   LIN {X -2.321, Y 6.996, Z 4.250} C_DIS
   LIN {X -2.151, Y 7.892, Z 4.250} C_DIS
   LIN {X -2.103, Y 8.164, Z 4.250} C_DIS
   LIN {X -1.982, Y 8.852, Z 4.250} C_DIS
   LIN {X -1.964, Y 8.960, Z 4.250} C_DIS
   LIN {X -1.822, Y 9.845, Z 4.250} C_DIS
   LIN {X -1.804, Y 9.955, Z 4.250} C_DIS
   LIN {X -1.672, Y 10.861, Z 4.250} C_DIS
   LIN {X -1.586, Y 11.505, Z 4.250} C_DIS
   LIN {X -1.538, Y 11.861, Z 4.250} C_DIS
   LIN {X -1.420, Y 12.858, Z 4.250} C_DIS
   LIN {X -1.315, Y 13.857, Z 4.250} C_DIS
   LIN {X -1.225, Y 14.841, Z 4.250} C_DIS
   LIN {X -1.150, Y 15.814, Z 4.250} C_DIS
   LIN {X -1.140, Y 15.955, Z 4.250} C_DIS
   LIN {X -1.088, Y 16.783, Z 4.250} C_DIS
   LIN {X -1.080, Y 16.934, Z 4.250} C_DIS
   LIN {X -1.038, Y 17.778, Z 4.250} C_DIS
   LIN {X -1.032, Y 17.929, Z 4.250} C_DIS
   LIN {X -1.001, Y 18.785, Z 4.250} C_DIS
   LIN {X -0.981, Y 19.646, Z 4.250} C_DIS
   LIN {X -0.976, Y 19.937, Z 4.250} C_DIS
   LIN {X -0.968, Y 20.790, Z 4.250} C_DIS
   LIN {X -0.969, Y 20.932, Z 4.250} C_DIS
   LIN {X -0.973, Y 21.776, Z 4.250} C_DIS
   LIN {X -0.975, Y 21.917, Z 4.250} C_DIS
   LIN {X -0.991, Y 22.780, Z 4.250} C_DIS
   LIN {X -0.995, Y 22.916, Z 4.250} C_DIS
   LIN {X -1.023, Y 23.792, Z 4.250} C_DIS
   LIN {X -1.029, Y 23.927, Z 4.250} C_DIS
   LIN {X -1.069, Y 24.801, Z 4.250} C_DIS
   LIN {X -1.077, Y 24.932, Z 4.250} C_DIS
   LIN {X -1.128, Y 25.791, Z 4.250} C_DIS
   LIN {X -1.137, Y 25.919, Z 4.250} C_DIS
   LIN {X -1.201, Y 26.794, Z 4.250} C_DIS
   LIN {X -1.212, Y 26.920, Z 4.250} C_DIS
   LIN {X -1.288, Y 27.797, Z 4.250} C_DIS
   LIN {X -1.301, Y 27.921, Z 4.250} C_DIS
   LIN {X -1.389, Y 28.791, Z 4.250} C_DIS
   LIN {X -1.402, Y 28.911, Z 4.250} C_DIS
   LIN {X -1.503, Y 29.784, Z 4.250} C_DIS
   LIN {X -1.517, Y 29.901, Z 4.250} C_DIS
   LIN {X -1.631, Y 30.783, Z 4.250} C_DIS
   LIN {X -1.646, Y 30.894, Z 4.250} C_DIS
   LIN {X -1.778, Y 31.812, Z 4.250} C_DIS
   LIN {X -1.870, Y 32.394, Z 4.250} C_DIS
   LIN {X -1.934, Y 32.804, Z 4.250} C_DIS
   LIN {X -1.964, Y 32.981, Z 4.250} C_DIS
   LIN {X -2.053, Y 33.505, Z 4.250} C_DIS
   LIN {X -2.116, Y 33.853, Z 4.250} C_DIS
   LIN {X -2.244, Y 34.558, Z 4.250} C_DIS
   LIN {X -2.371, Y 35.207, Z 4.250} C_DIS
   LIN {X -2.437, Y 35.536, Z 4.250} C_DIS
   LIN {X -2.623, Y 36.445, Z 4.250} C_DIS
   LIN {X -2.677, Y 36.710, Z 4.250} C_DIS
   LIN {X -2.693, Y 36.918, Z 4.250} C_DIS
   LIN {X -2.766, Y 37.917, Z 4.250} C_DIS
   LIN {X -2.645, Y 38.559, Z 4.250} C_DIS
   LIN {X -2.554, Y 38.861, Z 4.250} C_DIS
   LIN {X -2.172, Y 39.696, Z 4.250} C_DIS
   LIN {X -2.059, Y 39.830, Z 4.250} C_DIS
   LIN {X -1.515, Y 40.482, Z 4.250} C_DIS
   LIN {X -1.082, Y 40.815, Z 4.250} C_DIS
   LIN {X -0.713, Y 41.066, Z 4.250} C_DIS
   LIN {X -0.093, Y 41.307, Z 4.250} C_DIS
   LIN {X 0.221, Y 41.438, Z 4.250} C_DIS
   LIN {X 0.428, Y 41.467, Z 4.250} C_DIS
   LIN {X 1.905, Y 41.473, Z 4.250} C_DIS
   LIN {X 2.014, Y 41.460, Z 4.250} C_DIS
   LIN {X 2.928, Y 41.148, Z 4.250} C_DIS
   LIN {X 3.616, Y 40.710, Z 4.250} C_DIS
   LIN {X 3.955, Y 40.406, Z 4.250} C_DIS
   LIN {X 4.410, Y 39.919, Z 4.250} C_DIS
   LIN {X 4.780, Y 39.162, Z 4.250} C_DIS
   LIN {X 5.055, Y 38.597, Z 4.250} C_DIS
   LIN {X 5.286, Y 37.740, Z 4.250} C_DIS
   LIN {X 5.441, Y 37.175, Z 4.250} C_DIS
   LIN {X 5.746, Y 35.981, Z 4.250} C_DIS
   LIN {X 5.860, Y 35.543, Z 4.250} C_DIS
   LIN {X 6.103, Y 34.501, Z 4.250} C_DIS
   LIN {X 6.264, Y 33.837, Z 4.250} C_DIS
   LIN {X 6.422, Y 33.163, Z 4.250} C_DIS
   LIN {X 6.575, Y 32.475, Z 4.250} C_DIS
   LIN {X 6.724, Y 31.779, Z 4.250} C_DIS
   LIN {X 6.784, Y 31.497, Z 4.250} C_DIS
   LIN {X 6.926, Y 30.805, Z 4.250} C_DIS
   LIN {X 6.986, Y 30.510, Z 4.250} C_DIS
   LIN {X 7.126, Y 29.792, Z 4.250} C_DIS
   LIN {X 7.182, Y 29.506, Z 4.250} C_DIS
   LIN {X 7.313, Y 28.799, Z 4.250} C_DIS
   LIN {X 7.363, Y 28.527, Z 4.250} C_DIS
   LIN {X 7.486, Y 27.833, Z 4.250} C_DIS
   LIN {X 7.534, Y 27.558, Z 4.250} C_DIS
   LIN {X 7.652, Y 26.855, Z 4.250} C_DIS
   LIN {X 7.697, Y 26.581, Z 4.250} C_DIS
   LIN {X 7.809, Y 25.872, Z 4.250} C_DIS
   LIN {X 7.852, Y 25.599, Z 4.250} C_DIS
   LIN {X 7.960, Y 24.871, Z 4.250} C_DIS
   LIN {X 8.000, Y 24.599, Z 4.250} C_DIS
   LIN {X 8.102, Y 23.868, Z 4.250} C_DIS
   LIN {X 8.140, Y 23.596, Z 4.250} C_DIS
   LIN {X 8.234, Y 22.872, Z 4.250} C_DIS
   LIN {X 8.268, Y 22.612, Z 4.250} C_DIS
   LIN {X 8.354, Y 21.901, Z 4.250} C_DIS
   LIN {X 8.386, Y 21.636, Z 4.250} C_DIS
   LIN {X 8.469, Y 20.900, Z 4.250} C_DIS
   LIN {X 8.498, Y 20.638, Z 4.250} C_DIS
   LIN {X 8.572, Y 19.919, Z 4.250} C_DIS
   LIN {X 8.598, Y 19.667, Z 4.250} C_DIS
   LIN {X 8.668, Y 18.921, Z 4.250} C_DIS
   LIN {X 8.755, Y 17.912, Z 4.250} C_DIS
   LIN {X 8.766, Y 17.779, Z 4.250} C_DIS
   LIN {X 8.774, Y 17.677, Z 4.250} C_DIS
   LIN {X 8.851, Y 16.668, Z 4.250} C_DIS
   LIN {X 8.901, Y 15.921, Z 4.250} C_DIS
   LIN {X 8.917, Y 15.677, Z 4.250} C_DIS
   LIN {X 8.960, Y 14.935, Z 4.250} C_DIS
   LIN {X 8.974, Y 14.692, Z 4.250} C_DIS
   LIN {X 9.010, Y 13.941, Z 4.250} C_DIS
   LIN {X 9.022, Y 13.701, Z 4.250} C_DIS
   LIN {X 9.052, Y 12.932, Z 4.250} C_DIS
   LIN {X 9.061, Y 12.695, Z 4.250} C_DIS
   LIN {X 9.085, Y 11.925, Z 4.250} C_DIS
   LIN {X 9.091, Y 11.691, Z 4.250} C_DIS
   LIN {X 9.108, Y 10.928, Z 4.250} C_DIS
   LIN {X 9.112, Y 10.701, Z 4.250} C_DIS
   LIN {X 9.122, Y 9.945, Z 4.250} C_DIS
   LIN {X 9.124, Y 9.727, Z 4.250} C_DIS
   LIN {X 9.127, Y 8.959, Z 4.250} C_DIS
   LIN {X 9.127, Y 8.739, Z 4.250} C_DIS
   LIN {X 9.123, Y 7.966, Z 4.250} C_DIS
   LIN {X 9.121, Y 7.745, Z 4.250} C_DIS
   LIN {X 9.109, Y 6.932, Z 4.250} C_DIS
   LIN {X 9.106, Y 6.722, Z 4.250} C_DIS
   LIN {X 9.086, Y 5.918, Z 4.250} C_DIS
   LIN {X 9.081, Y 5.715, Z 4.250} C_DIS
   LIN {X 9.055, Y 4.933, Z 4.250} C_DIS
   LIN {X 9.048, Y 4.728, Z 4.250} C_DIS
   LIN {X 9.015, Y 3.957, Z 4.250} C_DIS
   LIN {X 9.006, Y 3.747, Z 4.250} C_DIS
   LIN {X 8.965, Y 2.958, Z 4.250} C_DIS
   LIN {X 8.954, Y 2.744, Z 4.250} C_DIS
   LIN {X 8.904, Y 1.935, Z 4.250} C_DIS
   LIN {X 8.891, Y 1.726, Z 4.250} C_DIS
   LIN {X 8.835, Y 0.921, Z 4.250} C_DIS
   LIN {X 8.820, Y 0.717, Z 4.250} C_DIS
   LIN {X 8.756, Y -0.090, Z 4.250} C_DIS
   LIN {X 8.740, Y -0.292, Z 4.250} C_DIS
   LIN {X 8.669, Y -1.088, Z 4.250} C_DIS
   LIN {X 8.639, Y -1.412, Z 4.250} C_DIS
   LIN {X 8.573, Y -2.092, Z 4.250} C_DIS
   LIN {X 8.495, Y -2.830, Z 4.250} C_DIS
   LIN {X 8.465, Y -3.107, Z 4.250} C_DIS
   LIN {X 8.350, Y -4.108, Z 4.250} C_DIS
   LIN {X 8.228, Y -5.092, Z 4.250} C_DIS
   LIN {X 8.214, Y -5.194, Z 4.250} C_DIS
   LIN {X 8.095, Y -6.086, Z 4.250} C_DIS
   LIN {X 8.080, Y -6.188, Z 4.250} C_DIS
   LIN {X 7.956, Y -7.059, Z 4.250} C_DIS
   LIN {X 7.940, Y -7.163, Z 4.250} C_DIS
   LIN {X 7.799, Y -8.086, Z 4.250} C_DIS
   LIN {X 7.712, Y -8.628, Z 4.250} C_DIS
   LIN {X 7.638, Y -9.084, Z 4.250} C_DIS
   LIN {X 7.487, Y -9.965, Z 4.250} C_DIS
   LIN {X 7.347, Y -10.745, Z 4.250} C_DIS
   LIN {X 7.304, Y -10.985, Z 4.250} C_DIS
   LIN {X 7.121, Y -11.952, Z 4.250} C_DIS
   LIN {X 7.091, Y -12.108, Z 4.250} C_DIS
   LIN {X 6.903, Y -13.044, Z 4.250} C_DIS
   LIN {X 6.872, Y -13.196, Z 4.250} C_DIS
   LIN {X 6.682, Y -14.099, Z 4.250} C_DIS
   LIN {X 6.650, Y -14.245, Z 4.250} C_DIS
   LIN {X 6.479, Y -15.028, Z 4.250} C_DIS
   LIN {X 6.450, Y -15.153, Z 4.250} C_DIS
   LIN {X 6.251, Y -16.024, Z 4.250} C_DIS
   LIN {X 6.221, Y -16.152, Z 4.250} C_DIS
   LIN {X 6.019, Y -16.997, Z 4.250} C_DIS
   LIN {X 5.988, Y -17.124, Z 4.250} C_DIS
   LIN {X 5.891, Y -17.511, Z 4.250} C_DIS
   LIN {X 5.744, Y -18.102, Z 4.250} C_DIS
   LIN {X 5.551, Y -18.849, Z 4.250} C_DIS
   LIN {X 5.486, Y -19.098, Z 4.250} C_DIS
   LIN {X 5.268, Y -19.909, Z 4.250} C_DIS
   LIN {X 5.229, Y -20.053, Z 4.250} C_DIS
   LIN {X 5.001, Y -20.872, Z 4.250} C_DIS
   LIN {X 4.961, Y -21.016, Z 4.250} C_DIS
   LIN {X 4.721, Y -21.846, Z 4.250} C_DIS
   LIN {X 4.514, Y -22.543, Z 4.250} C_DIS
   LIN {X 4.281, Y -23.311, Z 4.250} C_DIS
   LIN {X 4.231, Y -23.475, Z 4.250} C_DIS
   LIN {X 3.948, Y -24.383, Z 4.250} C_DIS
   LIN {X 3.631, Y -25.353, Z 4.250} C_DIS
   LIN {X 3.406, Y -26.038, Z 4.250} C_DIS
   LIN {X 3.244, Y -26.523, Z 4.250} C_DIS
   LIN {X 2.707, Y -27.741, Z 4.250} C_DIS
   LIN {X 2.623, Y -27.929, Z 4.250} C_DIS
   LIN {X 1.665, Y -29.352, Z 4.250} C_DIS
   LIN {X 0.963, Y -30.116, Z 4.250} C_DIS
   LIN {X 0.885, Y -30.181, Z 4.250} C_DIS
   LIN {X 0.158, Y -30.810, Z 4.250} C_DIS
   LIN {X -0.366, Y -31.180, Z 4.250} C_DIS
   LIN {X -0.678, Y -31.377, Z 4.250} C_DIS
   LIN {X -1.355, Y -31.750, Z 4.250} C_DIS
   LIN {X -1.553, Y -31.841, Z 4.250} C_DIS
   LIN {X -2.250, Y -32.132, Z 4.250} C_DIS
   LIN {X -2.473, Y -32.206, Z 4.250} C_DIS
   LIN {X -3.191, Y -32.419, Z 4.250} C_DIS
   LIN {X -3.426, Y -32.470, Z 4.250} C_DIS
   LIN {X -4.132, Y -32.600, Z 4.250} C_DIS
   LIN {X -4.382, Y -32.627, Z 4.250} C_DIS
   LIN {X -5.083, Y -32.679, Z 4.250} C_DIS
   LIN {X -5.347, Y -32.679, Z 4.250} C_DIS
   LIN {X -6.053, Y -32.655, Z 4.250} C_DIS
   LIN {X -6.333, Y -32.625, Z 4.250} C_DIS
   LIN {X -7.023, Y -32.526, Z 4.250} C_DIS
   LIN {X -7.296, Y -32.467, Z 4.250} C_DIS
   LIN {X -7.937, Y -32.304, Z 4.250} C_DIS
   LIN {X -8.216, Y -32.213, Z 4.250} C_DIS
   LIN {X -8.837, Y -31.982, Z 4.250} C_DIS
   LIN {X -9.120, Y -31.854, Z 4.250} C_DIS
   LIN {X -9.714, Y -31.556, Z 4.250} C_DIS
   LIN {X -9.967, Y -31.407, Z 4.250} C_DIS
   LIN {X -10.520, Y -31.049, Z 4.250} C_DIS
   LIN {X -10.759, Y -30.873, Z 4.250} C_DIS
   LIN {X -11.267, Y -30.460, Z 4.250} C_DIS
   LIN {X -11.502, Y -30.246, Z 4.250} C_DIS
   LIN {X -11.955, Y -29.789, Z 4.250}
   LaserEnd_Ext()
   LIN {X 7.602, Y -1.743, Z 4.250}
   LaserStart_Ext()
   LIN {X 7.602, Y 19.573, Z 4.250}
   LaserEnd_Ext()
   LIN {X 6.602, Y 27.068, Z 4.250}
   LaserStart_Ext()
   LIN {X 6.602, Y -9.210, Z 4.250}
   LaserEnd_Ext()
   LIN {X 5.602, Y -14.358, Z 4.250}
   LaserStart_Ext()
   LIN {X 5.602, Y 32.246, Z 4.250}
   LaserEnd_Ext()
   LIN {X 4.602, Y 36.418, Z 4.250}
   LaserStart_Ext()
   LIN {X 4.602, Y -18.524, Z 4.250}
   LaserEnd_Ext()
   LIN {X 3.602, Y -22.102, Z 4.250}
   LaserStart_Ext()
   LIN {X 3.602, Y 39.295, Z 4.250}
   LaserEnd_Ext()
   LIN {X 2.602, Y 40.170, Z 4.250}
   LaserStart_Ext()
   LIN {X 2.602, Y -25.281, Z 4.250}
   LaserEnd_Ext()
   LIN {X 1.602, Y -27.655, Z 4.250}
   LaserStart_Ext()
   LIN {X 1.602, Y 40.472, Z 4.250}
   LaserEnd_Ext()
   LIN {X 0.602, Y 40.468, Z 4.250}
   LaserStart_Ext()
   LIN {X 0.602, Y -29.032, Z 4.250}
   LaserEnd_Ext()
   LIN {X -0.398, Y -29.969, Z 4.250}
   LaserStart_Ext()
   LIN {X -0.398, Y 13.012, Z 4.250}
   LaserEnd_Ext()
   LIN {X -0.398, Y 28.931, Z 4.250}
   LaserStart_Ext()
   LIN {X -0.398, Y 40.070, Z 4.250}
   LaserEnd_Ext()
   LIN {X -1.398, Y 38.984, Z 4.250}
   LaserStart_Ext()
   LIN {X -1.398, Y 35.441, Z 4.250}
   LaserEnd_Ext()
   LIN {X -1.398, Y 6.512, Z 4.250}
   LaserStart_Ext()
   LIN {X -1.398, Y -30.632, Z 4.250}
   LaserEnd_Ext()
   LIN {X -2.398, Y -31.110, Z 4.250}
   LaserStart_Ext()
   LIN {X -2.398, Y 2.207, Z 4.250}
   LaserEnd_Ext()
   LIN {X -3.398, Y -1.228, Z 4.250}
   LaserStart_Ext()
   LIN {X -3.398, Y -31.437, Z 4.250}
   LaserEnd_Ext()
   LIN {X -4.398, Y -31.623, Z 4.250}
   LaserStart_Ext()
   LIN {X -4.398, Y -4.176, Z 4.250}
   LaserEnd_Ext()
   LIN {X -5.398, Y -6.767, Z 4.250}
   LaserStart_Ext()
   LIN {X -5.398, Y -31.677, Z 4.250}
   LaserEnd_Ext()
   LIN {X -6.398, Y -31.606, Z 4.250}
   LaserStart_Ext()
   LIN {X -6.398, Y -9.104, Z 4.250}
   LaserEnd_Ext()
   LIN {X -7.398, Y -11.243, Z 4.250}
   LaserStart_Ext()
   LIN {X -7.398, Y -31.409, Z 4.250}
   LaserEnd_Ext()
   LIN {X -8.398, Y -31.078, Z 4.250}
   LaserStart_Ext()
   LIN {X -8.398, Y -13.220, Z 4.250}
   LaserEnd_Ext()
   LIN {X -9.398, Y -15.058, Z 4.250}
   LaserStart_Ext()
   LIN {X -9.398, Y -30.582, Z 4.250}
   LaserEnd_Ext()
   LIN {X -10.398, Y -29.878, Z 4.250}
   LaserStart_Ext()
   LIN {X -10.398, Y -16.752, Z 4.250}
   LaserEnd_Ext()
   LIN {X -11.398, Y -18.400, Z 4.250}
   LaserStart_Ext()
   LIN {X -11.398, Y -28.909, Z 4.250}
   LaserEnd_Ext()
   LIN {X -12.398, Y -27.429, Z 4.250}
   LaserStart_Ext()
   LIN {X -12.398, Y -20.032, Z 4.250}
   LaserEnd_Ext()
   LIN {X -6.600, Y -7.105, Z 5.100}
   LaserStart_Ext()
   LIN {X -6.904, Y -7.825, Z 5.100} C_DIS
   LIN {X -6.989, Y -8.021, Z 5.100} C_DIS
   LIN {X -7.307, Y -8.745, Z 5.100} C_DIS
   LIN {X -7.394, Y -8.936, Z 5.100} C_DIS
   LIN {X -7.719, Y -9.650, Z 5.100} C_DIS
   LIN {X -7.806, Y -9.837, Z 5.100} C_DIS
   LIN {X -8.146, Y -10.556, Z 5.100} C_DIS
   LIN {X -8.236, Y -10.740, Z 5.100} C_DIS
   LIN {X -8.583, Y -11.451, Z 5.100} C_DIS
   LIN {X -8.675, Y -11.634, Z 5.100} C_DIS
   LIN {X -9.039, Y -12.351, Z 5.100} C_DIS
   LIN {X -9.132, Y -12.532, Z 5.100} C_DIS
   LIN {X -9.228, Y -12.710, Z 5.100} C_DIS
   LIN {X -9.326, Y -12.886, Z 5.100} C_DIS
   LIN {X -10.245, Y -14.598, Z 5.100} C_DIS
   LIN {X -11.082, Y -16.036, Z 5.100} C_DIS
   LIN {X -11.783, Y -17.211, Z 5.100} C_DIS
   LIN {X -12.498, Y -18.335, Z 5.100} C_DIS
   LIN {X -12.764, Y -18.757, Z 5.100} C_DIS
   LIN {X -12.941, Y -19.115, Z 5.100} C_DIS
   LIN {X -13.339, Y -19.810, Z 5.100} C_DIS
   LIN {X -13.777, Y -20.876, Z 5.100} C_DIS
   LIN {X -13.927, Y -22.331, Z 5.100} C_DIS
   LIN {X -14.210, Y -24.293, Z 5.100} C_DIS
   LIN {X -14.150, Y -24.896, Z 5.100} C_DIS
   LIN {X -13.983, Y -25.790, Z 5.100} C_DIS
   LIN {X -13.959, Y -25.887, Z 5.100} C_DIS
   LIN {X -13.706, Y -26.718, Z 5.100} C_DIS
   LIN {X -13.342, Y -27.587, Z 5.100} C_DIS
   LIN {X -12.867, Y -28.450, Z 5.100} C_DIS
   LIN {X -12.813, Y -28.536, Z 5.100} C_DIS
   LIN {X -12.325, Y -29.221, Z 5.100} C_DIS
   LIN {X -12.262, Y -29.300, Z 5.100} C_DIS
   LIN {X -11.705, Y -29.930, Z 5.100} C_DIS
   LIN {X -10.998, Y -30.582, Z 5.100} C_DIS
   LIN {X -10.913, Y -30.651, Z 5.100} C_DIS
   LIN {X -10.255, Y -31.137, Z 5.100} C_DIS
   LIN {X -10.158, Y -31.199, Z 5.100} C_DIS
   LIN {X -9.456, Y -31.612, Z 5.100} C_DIS
   LIN {X -9.351, Y -31.665, Z 5.100} C_DIS
   LIN {X -8.568, Y -32.018, Z 5.100} C_DIS
   LIN {X -8.462, Y -32.058, Z 5.100} C_DIS
   LIN {X -7.676, Y -32.315, Z 5.100} C_DIS
   LIN {X -7.554, Y -32.346, Z 5.100} C_DIS
   LIN {X -6.758, Y -32.518, Z 5.100} C_DIS
   LIN {X -6.617, Y -32.538, Z 5.100} C_DIS
   LIN {X -5.785, Y -32.627, Z 5.100} C_DIS
   LIN {X -5.635, Y -32.632, Z 5.100} C_DIS
   LIN {X -4.835, Y -32.631, Z 5.100} C_DIS
   LIN {X -4.674, Y -32.619, Z 5.100} C_DIS
   LIN {X -3.892, Y -32.534, Z 5.100} C_DIS
   LIN {X -3.721, Y -32.503, Z 5.100} C_DIS
   LIN {X -2.954, Y -32.337, Z 5.100} C_DIS
   LIN {X -2.770, Y -32.282, Z 5.100} C_DIS
   LIN {X -2.018, Y -32.033, Z 5.100} C_DIS
   LIN {X -1.833, Y -31.955, Z 5.100} C_DIS
   LIN {X -1.127, Y -31.634, Z 5.100} C_DIS
   LIN {X -0.937, Y -31.529, Z 5.100} C_DIS
   LIN {X -0.468, Y -31.232, Z 5.100} C_DIS
   LIN {X 0.129, Y -30.849, Z 5.100} C_DIS
   LIN {X 0.841, Y -30.256, Z 5.100} C_DIS
   LIN {X 1.255, Y -29.807, Z 5.100} C_DIS
   LIN {X 2.061, Y -28.862, Z 5.100} C_DIS
   LIN {X 2.631, Y -28.015, Z 5.100} C_DIS
   LIN {X 3.177, Y -26.794, Z 5.100} C_DIS
   LIN {X 3.330, Y -26.460, Z 5.100} C_DIS
   LIN {X 3.482, Y -25.992, Z 5.100} C_DIS
   LIN {X 3.825, Y -24.949, Z 5.100} C_DIS
   LIN {X 3.984, Y -24.461, Z 5.100} C_DIS
   LIN {X 4.127, Y -24.005, Z 5.100} C_DIS
   LIN {X 4.408, Y -23.079, Z 5.100} C_DIS
   LIN {X 4.704, Y -22.078, Z 5.100} C_DIS
   LIN {X 4.782, Y -21.821, Z 5.100} C_DIS
   LIN {X 4.851, Y -21.587, Z 5.100} C_DIS
   LIN {X 4.932, Y -21.309, Z 5.100} C_DIS
   LIN {X 5.127, Y -20.611, Z 5.100} C_DIS
   LIN {X 5.203, Y -20.338, Z 5.100} C_DIS
   LIN {X 5.390, Y -19.647, Z 5.100} C_DIS
   LIN {X 5.462, Y -19.378, Z 5.100} C_DIS
   LIN {X 5.676, Y -18.555, Z 5.100} C_DIS
   LIN {X 5.747, Y -18.278, Z 5.100} C_DIS
   LIN {X 5.824, Y -17.965, Z 5.100} C_DIS
   LIN {X 6.066, Y -16.989, Z 5.100} C_DIS
   LIN {X 6.149, Y -16.644, Z 5.100} C_DIS
   LIN {X 6.328, Y -15.876, Z 5.100} C_DIS
   LIN {X 6.456, Y -15.316, Z 5.100} C_DIS
   LIN {X 6.555, Y -14.865, Z 5.100} C_DIS
   LIN {X 6.661, Y -14.383, Z 5.100} C_DIS
   LIN {X 6.779, Y -13.826, Z 5.100} C_DIS
   LIN {X 6.860, Y -13.439, Z 5.100} C_DIS
   LIN {X 6.995, Y -12.770, Z 5.100} C_DIS
   LIN {X 7.057, Y -12.461, Z 5.100} C_DIS
   LIN {X 7.208, Y -11.677, Z 5.100} C_DIS
   LIN {X 7.272, Y -11.338, Z 5.100} C_DIS
   LIN {X 7.524, Y -9.916, Z 5.100} C_DIS
   LIN {X 7.573, Y -9.642, Z 5.100} C_DIS
   LIN {X 7.624, Y -9.344, Z 5.100} C_DIS
   LIN {X 7.711, Y -8.812, Z 5.100} C_DIS
   LIN {X 7.778, Y -8.399, Z 5.100} C_DIS
   LIN {X 7.862, Y -7.851, Z 5.100} C_DIS
   LIN {X 7.936, Y -7.366, Z 5.100} C_DIS
   LIN {X 8.005, Y -6.889, Z 5.100} C_DIS
   LIN {X 8.080, Y -6.364, Z 5.100} C_DIS
   LIN {X 8.141, Y -5.907, Z 5.100} C_DIS
   LIN {X 8.213, Y -5.372, Z 5.100} C_DIS
   LIN {X 8.271, Y -4.908, Z 5.100} C_DIS
   LIN {X 8.337, Y -4.382, Z 5.100} C_DIS
   LIN {X 8.390, Y -3.920, Z 5.100} C_DIS
   LIN {X 8.452, Y -3.388, Z 5.100} C_DIS
   LIN {X 8.572, Y -2.236, Z 5.100} C_DIS
   LIN {X 8.599, Y -1.980, Z 5.100} C_DIS
   LIN {X 8.642, Y -1.507, Z 5.100} C_DIS
   LIN {X 8.707, Y -0.804, Z 5.100} C_DIS
   LIN {X 8.728, Y -0.570, Z 5.100} C_DIS
   LIN {X 8.790, Y 0.199, Z 5.100} C_DIS
   LIN {X 8.809, Y 0.434, Z 5.100} C_DIS
   LIN {X 8.864, Y 1.207, Z 5.100} C_DIS
   LIN {X 8.880, Y 1.439, Z 5.100} C_DIS
   LIN {X 8.929, Y 2.221, Z 5.100} C_DIS
   LIN {X 8.943, Y 2.452, Z 5.100} C_DIS
   LIN {X 8.985, Y 3.244, Z 5.100} C_DIS
   LIN {X 8.997, Y 3.467, Z 5.100} C_DIS
   LIN {X 9.030, Y 4.240, Z 5.100} C_DIS
   LIN {X 9.039, Y 4.456, Z 5.100} C_DIS
   LIN {X 9.066, Y 5.216, Z 5.100} C_DIS
   LIN {X 9.073, Y 5.437, Z 5.100} C_DIS
   LIN {X 9.093, Y 6.201, Z 5.100} C_DIS
   LIN {X 9.098, Y 6.432, Z 5.100} C_DIS
   LIN {X 9.111, Y 7.216, Z 5.100} C_DIS
   LIN {X 9.114, Y 7.447, Z 5.100} C_DIS
   LIN {X 9.120, Y 8.249, Z 5.100} C_DIS
   LIN {X 9.121, Y 8.464, Z 5.100} C_DIS
   LIN {X 9.120, Y 9.256, Z 5.100} C_DIS
   LIN {X 9.119, Y 9.464, Z 5.100} C_DIS
   LIN {X 9.110, Y 10.219, Z 5.100} C_DIS
   LIN {X 9.108, Y 10.421, Z 5.100} C_DIS
   LIN {X 9.092, Y 11.202, Z 5.100} C_DIS
   LIN {X 9.088, Y 11.404, Z 5.100} C_DIS
   LIN {X 9.064, Y 12.217, Z 5.100} C_DIS
   LIN {X 9.058, Y 12.421, Z 5.100} C_DIS
   LIN {X 9.027, Y 13.224, Z 5.100} C_DIS
   LIN {X 9.020, Y 13.422, Z 5.100} C_DIS
   LIN {X 8.981, Y 14.226, Z 5.100} C_DIS
   LIN {X 8.972, Y 14.415, Z 5.100} C_DIS
   LIN {X 8.927, Y 15.219, Z 5.100} C_DIS
   LIN {X 8.916, Y 15.404, Z 5.100} C_DIS
   LIN {X 8.864, Y 16.205, Z 5.100} C_DIS
   LIN {X 8.851, Y 16.389, Z 5.100} C_DIS
   LIN {X 8.829, Y 16.684, Z 5.100} C_DIS
   LIN {X 8.744, Y 17.797, Z 5.100} C_DIS
   LIN {X 8.642, Y 18.919, Z 5.100} C_DIS
   LIN {X 8.617, Y 19.206, Z 5.100} C_DIS
   LIN {X 8.600, Y 19.385, Z 5.100} C_DIS
   LIN {X 8.519, Y 20.186, Z 5.100} C_DIS
   LIN {X 8.501, Y 20.357, Z 5.100} C_DIS
   LIN {X 8.409, Y 21.182, Z 5.100} C_DIS
   LIN {X 8.390, Y 21.353, Z 5.100} C_DIS
   LIN {X 8.291, Y 22.182, Z 5.100} C_DIS
   LIN {X 8.271, Y 22.343, Z 5.100} C_DIS
   LIN {X 8.167, Y 23.153, Z 5.100} C_DIS
   LIN {X 8.146, Y 23.315, Z 5.100} C_DIS
   LIN {X 8.029, Y 24.156, Z 5.100} C_DIS
   LIN {X 8.007, Y 24.319, Z 5.100} C_DIS
   LIN {X 7.884, Y 25.154, Z 5.100} C_DIS
   LIN {X 7.860, Y 25.314, Z 5.100} C_DIS
   LIN {X 7.729, Y 26.151, Z 5.100} C_DIS
   LIN {X 7.704, Y 26.305, Z 5.100} C_DIS
   LIN {X 7.567, Y 27.132, Z 5.100} C_DIS
   LIN {X 7.542, Y 27.281, Z 5.100} C_DIS
   LIN {X 7.398, Y 28.106, Z 5.100} C_DIS
   LIN {X 7.372, Y 28.249, Z 5.100} C_DIS
   LIN {X 7.224, Y 29.056, Z 5.100} C_DIS
   LIN {X 7.196, Y 29.204, Z 5.100} C_DIS
   LIN {X 7.033, Y 30.048, Z 5.100} C_DIS
   LIN {X 7.004, Y 30.196, Z 5.100} C_DIS
   LIN {X 6.829, Y 31.060, Z 5.100} C_DIS
   LIN {X 6.800, Y 31.201, Z 5.100} C_DIS
   LIN {X 6.621, Y 32.043, Z 5.100} C_DIS
   LIN {X 6.592, Y 32.179, Z 5.100} C_DIS
   LIN {X 6.562, Y 32.313, Z 5.100} C_DIS
   LIN {X 6.531, Y 32.444, Z 5.100} C_DIS
   LIN {X 6.500, Y 32.574, Z 5.100} C_DIS
   LIN {X 5.812, Y 35.528, Z 5.100} C_DIS
   LIN {X 5.487, Y 36.770, Z 5.100} C_DIS
   LIN {X 5.368, Y 37.235, Z 5.100} C_DIS
   LIN {X 5.155, Y 38.017, Z 5.100} C_DIS
   LIN {X 4.977, Y 38.664, Z 5.100} C_DIS
   LIN {X 4.582, Y 39.467, Z 5.100} C_DIS
   LIN {X 4.329, Y 39.985, Z 5.100} C_DIS
   LIN {X 4.214, Y 40.108, Z 5.100} C_DIS
   LIN {X 3.291, Y 40.938, Z 5.100} C_DIS
   LIN {X 2.923, Y 41.172, Z 5.100} C_DIS
   LIN {X 2.395, Y 41.352, Z 5.100} C_DIS
   LIN {X 1.670, Y 41.556, Z 5.100} C_DIS
   LIN {X 0.602, Y 41.542, Z 5.100} C_DIS
   LIN {X -0.338, Y 41.323, Z 5.100} C_DIS
   LIN {X -0.622, Y 41.213, Z 5.100} C_DIS
   LIN {X -1.002, Y 40.954, Z 5.100} C_DIS
   LIN {X -1.393, Y 40.705, Z 5.100} C_DIS
   LIN {X -1.963, Y 40.071, Z 5.100} C_DIS
   LIN {X -2.300, Y 39.670, Z 5.100} C_DIS
   LIN {X -2.389, Y 39.476, Z 5.100} C_DIS
   LIN {X -2.690, Y 38.477, Z 5.100} C_DIS
   LIN {X -2.837, Y 38.032, Z 5.100} C_DIS
   LIN {X -2.828, Y 37.850, Z 5.100} C_DIS
   LIN {X -2.751, Y 36.759, Z 5.100} C_DIS
   LIN {X -2.527, Y 35.676, Z 5.100} C_DIS
   LIN {X -2.499, Y 35.539, Z 5.100} C_DIS
   LIN {X -2.317, Y 34.622, Z 5.100} C_DIS
   LIN {X -2.293, Y 34.494, Z 5.100} C_DIS
   LIN {X -2.198, Y 33.963, Z 5.100} C_DIS
   LIN {X -2.033, Y 33.050, Z 5.100} C_DIS
   LIN {X -1.956, Y 32.579, Z 5.100} C_DIS
   LIN {X -1.858, Y 31.957, Z 5.100} C_DIS
   LIN {X -1.789, Y 31.520, Z 5.100} C_DIS
   LIN {X -1.735, Y 31.143, Z 5.100} C_DIS
   LIN {X -1.644, Y 30.491, Z 5.100} C_DIS
   LIN {X -1.603, Y 30.172, Z 5.100} C_DIS
   LIN {X -1.519, Y 29.496, Z 5.100} C_DIS
   LIN {X -1.483, Y 29.181, Z 5.100} C_DIS
   LIN {X -1.407, Y 28.503, Z 5.100} C_DIS
   LIN {X -1.376, Y 28.190, Z 5.100} C_DIS
   LIN {X -1.309, Y 27.503, Z 5.100} C_DIS
   LIN {X -1.281, Y 27.190, Z 5.100} C_DIS
   LIN {X -1.224, Y 26.505, Z 5.100} C_DIS
   LIN {X -1.202, Y 26.194, Z 5.100} C_DIS
   LIN {X -1.154, Y 25.506, Z 5.100} C_DIS
   LIN {X -1.135, Y 25.203, Z 5.100} C_DIS
   LIN {X -1.097, Y 24.511, Z 5.100} C_DIS
   LIN {X -1.083, Y 24.204, Z 5.100} C_DIS
   LIN {X -1.053, Y 23.501, Z 5.100} C_DIS
   LIN {X -1.043, Y 23.195, Z 5.100} C_DIS
   LIN {X -1.023, Y 22.498, Z 5.100} C_DIS
   LIN {X -1.018, Y 22.199, Z 5.100} C_DIS
   LIN {X -1.007, Y 21.495, Z 5.100} C_DIS
   LIN {X -1.006, Y 21.204, Z 5.100} C_DIS
   LIN {X -1.005, Y 20.501, Z 5.100} C_DIS
   LIN {X -1.008, Y 20.208, Z 5.100} C_DIS
   LIN {X -1.035, Y 18.794, Z 5.100} C_DIS
   LIN {X -1.042, Y 18.502, Z 5.100} C_DIS
   LIN {X -1.052, Y 18.212, Z 5.100} C_DIS
   LIN {X -1.081, Y 17.495, Z 5.100} C_DIS
   LIN {X -1.095, Y 17.211, Z 5.100} C_DIS
   LIN {X -1.132, Y 16.509, Z 5.100} C_DIS
   LIN {X -1.150, Y 16.232, Z 5.100} C_DIS
   LIN {X -1.193, Y 15.583, Z 5.100} C_DIS
   LIN {X -1.219, Y 15.253, Z 5.100} C_DIS
   LIN {X -1.266, Y 14.652, Z 5.100} C_DIS
   LIN {X -1.302, Y 14.264, Z 5.100} C_DIS
   LIN {X -1.358, Y 13.658, Z 5.100} C_DIS
   LIN {X -1.399, Y 13.267, Z 5.100} C_DIS
   LIN {X -1.462, Y 12.668, Z 5.100} C_DIS
   LIN {X -1.511, Y 12.259, Z 5.100} C_DIS
   LIN {X -1.581, Y 11.679, Z 5.100} C_DIS
   LIN {X -1.640, Y 11.236, Z 5.100} C_DIS
   LIN {X -1.723, Y 10.624, Z 5.100} C_DIS
   LIN {X -1.795, Y 10.134, Z 5.100} C_DIS
   LIN {X -1.864, Y 9.674, Z 5.100} C_DIS
   LIN {X -1.951, Y 9.129, Z 5.100} C_DIS
   LIN {X -2.029, Y 8.659, Z 5.100} C_DIS
   LIN {X -2.112, Y 8.184, Z 5.100} C_DIS
   LIN {X -2.216, Y 7.607, Z 5.100} C_DIS
   LIN {X -2.286, Y 7.234, Z 5.100} C_DIS
   LIN {X -2.421, Y 6.541, Z 5.100} C_DIS
   LIN {X -2.472, Y 6.296, Z 5.100} C_DIS
   LIN {X -2.623, Y 5.574, Z 5.100} C_DIS
   LIN {X -2.678, Y 5.324, Z 5.100} C_DIS
   LIN {X -2.844, Y 4.582, Z 5.100} C_DIS
   LIN {X -2.902, Y 4.333, Z 5.100} C_DIS
   LIN {X -3.079, Y 3.593, Z 5.100} C_DIS
   LIN {X -3.139, Y 3.352, Z 5.100} C_DIS
   LIN {X -3.204, Y 3.103, Z 5.100} C_DIS
   LIN {X -3.504, Y 1.943, Z 5.100} C_DIS
   LIN {X -3.724, Y 1.156, Z 5.100} C_DIS
   LIN {X -4.174, Y -0.376, Z 5.100} C_DIS
   LIN {X -4.249, Y -0.628, Z 5.100} C_DIS
   LIN {X -4.309, Y -0.815, Z 5.100} C_DIS
   LIN {X -4.759, Y -2.208, Z 5.100} C_DIS
   LIN {X -4.833, Y -2.426, Z 5.100} C_DIS
   LIN {X -5.086, Y -3.161, Z 5.100} C_DIS
   LIN {X -5.160, Y -3.371, Z 5.100} C_DIS
   LIN {X -5.418, Y -4.087, Z 5.100} C_DIS
   LIN {X -5.494, Y -4.294, Z 5.100} C_DIS
   LIN {X -5.764, Y -5.015, Z 5.100} C_DIS
   LIN {X -5.844, Y -5.221, Z 5.100} C_DIS
   LIN {X -6.129, Y -5.951, Z 5.100} C_DIS
   LIN {X -6.213, Y -6.160, Z 5.100} C_DIS
   LIN {X -6.515, Y -6.903, Z 5.100} C_DIS
   LIN {X -6.600, Y -7.105, Z 5.100}
   LaserEnd_Ext()
   LIN {X 1.654, Y 40.522, Z 5.100}
   LaserStart_Ext()
   LIN {X 0.629, Y 40.522, Z 5.100}
   LaserEnd_Ext()
   LIN {X -1.112, Y 39.522, Z 5.100}
   LaserStart_Ext()
   LIN {X 3.370, Y 39.522, Z 5.100}
   LaserEnd_Ext()
   LIN {X 3.933, Y 38.522, Z 5.100}
   LaserStart_Ext()
   LIN {X -1.632, Y 38.522, Z 5.100}
   LaserEnd_Ext()
   LIN {X -1.803, Y 37.522, Z 5.100}
   LaserStart_Ext()
   LIN {X 4.253, Y 37.522, Z 5.100}
   LaserEnd_Ext()
   LIN {X 4.518, Y 36.522, Z 5.100}
   LaserStart_Ext()
   LIN {X -1.681, Y 36.522, Z 5.100}
   LaserEnd_Ext()
   LIN {X -1.476, Y 35.522, Z 5.100}
   LaserStart_Ext()
   LIN {X 4.780, Y 35.522, Z 5.100}
   LaserEnd_Ext()
   LIN {X 5.019, Y 34.522, Z 5.100}
   LaserStart_Ext()
   LIN {X -1.282, Y 34.522, Z 5.100}
   LaserEnd_Ext()
   LIN {X -1.102, Y 33.522, Z 5.100}
   LaserStart_Ext()
   LIN {X 5.252, Y 33.522, Z 5.100}
   LaserEnd_Ext()
   LIN {X 5.485, Y 32.522, Z 5.100}
   LaserStart_Ext()
   LIN {X -0.935, Y 32.522, Z 5.100}
   LaserEnd_Ext()
   LIN {X -0.779, Y 31.522, Z 5.100}
   LaserStart_Ext()
   LIN {X 5.709, Y 31.522, Z 5.100}
   LaserEnd_Ext()
   LIN {X 5.918, Y 30.522, Z 5.100}
   LaserStart_Ext()
   LIN {X -0.640, Y 30.522, Z 5.100}
   LaserEnd_Ext()
   LIN {X -0.515, Y 29.522, Z 5.100}
   LaserStart_Ext()
   LIN {X 6.116, Y 29.522, Z 5.100}
   LaserEnd_Ext()
   LIN {X 6.305, Y 28.522, Z 5.100}
   LaserStart_Ext()
   LIN {X -0.404, Y 28.522, Z 5.100}
   LaserEnd_Ext()
   LIN {X -0.307, Y 27.522, Z 5.100}
   LaserStart_Ext()
   LIN {X 6.485, Y 27.522, Z 5.100}
   LaserEnd_Ext()
   LIN {X 6.654, Y 26.522, Z 5.100}
   LaserStart_Ext()
   LIN {X -0.223, Y 26.522, Z 5.100}
   LaserEnd_Ext()
   LIN {X -0.153, Y 25.522, Z 5.100}
   LaserStart_Ext()
   LIN {X 6.815, Y 25.522, Z 5.100}
   LaserEnd_Ext()
   LIN {X 6.966, Y 24.522, Z 5.100}
   LaserStart_Ext()
   LIN {X -0.096, Y 24.522, Z 5.100}
   LaserEnd_Ext()
   LIN {X -0.053, Y 23.522, Z 5.100}
   LaserStart_Ext()
   LIN {X 7.108, Y 23.522, Z 5.100}
   LaserEnd_Ext()
   LIN {X 7.240, Y 22.522, Z 5.100}
   LaserStart_Ext()
   LIN {X -0.024, Y 22.522, Z 5.100}
   LaserEnd_Ext()
   LIN {X -0.008, Y 21.522, Z 5.100}
   LaserStart_Ext()
   LIN {X 7.363, Y 21.522, Z 5.100}
   LaserEnd_Ext()
   LIN {X 7.477, Y 20.522, Z 5.100}
   LaserStart_Ext()
   LIN {X -0.005, Y 20.522, Z 5.100}
   LaserEnd_Ext()
   LIN {X -0.021, Y 19.522, Z 5.100}
   LaserStart_Ext()
   LIN {X 7.581, Y 19.522, Z 5.100}
   LaserEnd_Ext()
   LIN {X 7.674, Y 18.522, Z 5.100}
   LaserStart_Ext()
   LIN {X -0.041, Y 18.522, Z 5.100}
   LaserEnd_Ext()
   LIN {X -0.079, Y 17.522, Z 5.100}
   LaserStart_Ext()
   LIN {X 7.762, Y 17.522, Z 5.100}
   LaserEnd_Ext()
   LIN {X 7.838, Y 16.522, Z 5.100}
   LaserStart_Ext()
   LIN {X -0.130, Y 16.522, Z 5.100}
   LaserEnd_Ext()
   LIN {X -0.195, Y 15.522, Z 5.100}
   LaserStart_Ext()
   LIN {X 7.906, Y 15.522, Z 5.100}
   LaserEnd_Ext()
   LIN {X 7.965, Y 14.522, Z 5.100}
   LaserStart_Ext()
   LIN {X -0.274, Y 14.522, Z 5.100}
   LaserEnd_Ext()
   LIN {X -0.367, Y 13.522, Z 5.100}
   LaserStart_Ext()
   LIN {X 8.014, Y 13.522, Z 5.100}
   LaserEnd_Ext()
   LIN {X 8.054, Y 12.522, Z 5.100}
   LaserStart_Ext()
   LIN {X -0.473, Y 12.522, Z 5.100}
   LaserEnd_Ext()
   LIN {X -0.593, Y 11.522, Z 5.100}
   LaserStart_Ext()
   LIN {X 8.084, Y 11.522, Z 5.100}
   LaserEnd_Ext()
   LIN {X 8.106, Y 10.522, Z 5.100}
   LaserStart_Ext()
   LIN {X -0.727, Y 10.522, Z 5.100}
   LaserEnd_Ext()
   LIN {X -0.875, Y 9.522, Z 5.100}
   LaserStart_Ext()
   LIN {X 8.118, Y 9.522, Z 5.100}
   LaserEnd_Ext()
   LIN {X 8.121, Y 8.522, Z 5.100}
   LaserStart_Ext()
   LIN {X -1.038, Y 8.522, Z 5.100}
   LaserEnd_Ext()
   LIN {X -1.215, Y 7.522, Z 5.100}
   LaserStart_Ext()
   LIN {X 8.115, Y 7.522, Z 5.100}
   LaserEnd_Ext()
   LIN {X 8.100, Y 6.522, Z 5.100}
   LaserStart_Ext()
   LIN {X -1.407, Y 6.522, Z 5.100}
   LaserEnd_Ext()
   LIN {X -1.612, Y 5.522, Z 5.100}
   LaserStart_Ext()
   LIN {X 8.075, Y 5.522, Z 5.100}
   LaserEnd_Ext()
   LIN {X 8.041, Y 4.522, Z 5.100}
   LaserStart_Ext()
   LIN {X -1.833, Y 4.522, Z 5.100}
   LaserEnd_Ext()
   LIN {X -2.068, Y 3.522, Z 5.100}
   LaserStart_Ext()
   LIN {X 7.998, Y 3.522, Z 5.100}
   LaserEnd_Ext()
   LIN {X 7.945, Y 2.522, Z 5.100}
   LaserStart_Ext()
   LIN {X -2.321, Y 2.522, Z 5.100}
   LaserEnd_Ext()
   LIN {X -2.583, Y 1.522, Z 5.100}
   LaserStart_Ext()
   LIN {X 7.884, Y 1.522, Z 5.100}
   LaserEnd_Ext()
   LIN {X 7.813, Y 0.522, Z 5.100}
   LaserStart_Ext()
   LIN {X -2.868, Y 0.522, Z 5.100}
   LaserEnd_Ext()
   LIN {X -3.161, Y -0.478, Z 5.100}
   LaserStart_Ext()
   LIN {X 7.732, Y -0.478, Z 5.100}
   LaserEnd_Ext()
   LIN {X 7.641, Y -1.478, Z 5.100}
   LaserStart_Ext()
   LIN {X -3.472, Y -1.478, Z 5.100}
   LaserEnd_Ext()
   LIN {X -3.795, Y -2.478, Z 5.100}
   LaserStart_Ext()
   LIN {X 7.541, Y -2.478, Z 5.100}
   LaserEnd_Ext()
   LIN {X 7.435, Y -3.478, Z 5.100}
   LaserStart_Ext()
   LIN {X -4.137, Y -3.478, Z 5.100}
   LaserEnd_Ext()
   LIN {X -4.496, Y -4.478, Z 5.100}
   LaserStart_Ext()
   LIN {X 7.317, Y -4.478, Z 5.100}
   LaserEnd_Ext()
   LIN {X 7.190, Y -5.478, Z 5.100}
   LaserStart_Ext()
   LIN {X -4.871, Y -5.478, Z 5.100}
   LaserEnd_Ext()
   LIN {X -5.263, Y -6.478, Z 5.100}
   LaserStart_Ext()
   LIN {X 7.053, Y -6.478, Z 5.100}
   LaserEnd_Ext()
   LIN {X 6.907, Y -7.478, Z 5.100}
   LaserStart_Ext()
   LIN {X -5.672, Y -7.478, Z 5.100}
   LaserEnd_Ext()
   LIN {X -6.098, Y -8.478, Z 5.100}
   LaserStart_Ext()
   LIN {X 6.752, Y -8.478, Z 5.100}
   LaserEnd_Ext()
   LIN {X 6.586, Y -9.478, Z 5.100}
   LaserStart_Ext()
   LIN {X -6.542, Y -9.478, Z 5.100}
   LaserEnd_Ext()
   LIN {X -7.004, Y -10.478, Z 5.100}
   LaserStart_Ext()
   LIN {X 6.409, Y -10.478, Z 5.100}
   LaserEnd_Ext()
   LIN {X 6.228, Y -11.478, Z 5.100}
   LaserStart_Ext()
   LIN {X -7.483, Y -11.478, Z 5.100}
   LaserEnd_Ext()
   LIN {X -7.982, Y -12.478, Z 5.100}
   LaserStart_Ext()
   LIN {X 6.034, Y -12.478, Z 5.100}
   LaserEnd_Ext()
   LIN {X 5.830, Y -13.478, Z 5.100}
   LaserStart_Ext()
   LIN {X -8.509, Y -13.478, Z 5.100}
   LaserEnd_Ext()
   LIN {X -9.046, Y -14.478, Z 5.100}
   LaserStart_Ext()
   LIN {X 5.616, Y -14.478, Z 5.100}
   LaserEnd_Ext()
   LIN {X 5.393, Y -15.478, Z 5.100}
   LaserStart_Ext()
   LIN {X -9.600, Y -15.478, Z 5.100}
   LaserEnd_Ext()
   LIN {X -10.182, Y -16.478, Z 5.100}
   LaserStart_Ext()
   LIN {X 5.160, Y -16.478, Z 5.100}
   LaserEnd_Ext()
   LIN {X 4.915, Y -17.478, Z 5.100}
   LaserStart_Ext()
   LIN {X -10.778, Y -17.478, Z 5.100}
   LaserEnd_Ext()
   LIN {X -11.404, Y -18.478, Z 5.100}
   LaserStart_Ext()
   LIN {X 4.662, Y -18.478, Z 5.100}
   LaserEnd_Ext()
   LIN {X 4.400, Y -19.478, Z 5.100}
   LaserStart_Ext()
   LIN {X -12.005, Y -19.478, Z 5.100}
   LaserEnd_Ext()
   LIN {X -12.532, Y -20.478, Z 5.100}
   LaserStart_Ext()
   LIN {X 4.126, Y -20.478, Z 5.100}
   LaserEnd_Ext()
   LIN {X 3.841, Y -21.478, Z 5.100}
   LaserStart_Ext()
   LIN {X -12.834, Y -21.478, Z 5.100}
   LaserEnd_Ext()
   LIN {X -12.938, Y -22.478, Z 5.100}
   LaserStart_Ext()
   LIN {X 3.543, Y -22.478, Z 5.100}
   LaserEnd_Ext()
   LIN {X 3.241, Y -23.478, Z 5.100}
   LaserStart_Ext()
   LIN {X -13.082, Y -23.478, Z 5.100}
   LaserEnd_Ext()
   LIN {X -13.187, Y -24.478, Z 5.100}
   LaserStart_Ext()
   LIN {X 2.926, Y -24.478, Z 5.100}
   LaserEnd_Ext()
   LIN {X 2.598, Y -25.478, Z 5.100}
   LaserStart_Ext()
   LIN {X -13.025, Y -25.478, Z 5.100}
   LaserEnd_Ext()
   LIN {X -12.727, Y -26.478, Z 5.100}
   LaserStart_Ext()
   LIN {X 2.222, Y -26.478, Z 5.100}
   LaserEnd_Ext()
   LIN {X 1.776, Y -27.478, Z 5.100}
   LaserStart_Ext()
   LIN {X -12.264, Y -27.478, Z 5.100}
   LaserEnd_Ext()
   LIN {X -11.627, Y -28.478, Z 5.100}
   LaserStart_Ext()
   LIN {X 1.074, Y -28.478, Z 5.100}
   LaserEnd_Ext()
   LIN {X 0.198, Y -29.478, Z 5.100}
   LaserStart_Ext()
   LIN {X -10.724, Y -29.478, Z 5.100}
   LaserEnd_Ext()
   LIN {X -9.411, Y -30.478, Z 5.100}
   LaserStart_Ext()
   LIN {X -1.147, Y -30.478, Z 5.100}
   LaserEnd_Ext()
   LIN {X -3.714, Y -31.478, Z 5.100}
   LaserStart_Ext()
   LIN {X -6.834, Y -31.478, Z 5.100}
   LaserEnd_Ext()
   LIN {X 9.017, Y 13.187, Z 5.950}
   LaserStart_Ext()
   LIN {X 9.004, Y 13.471, Z 5.950} C_DIS
   LIN {X 8.970, Y 14.180, Z 5.950} C_DIS
   LIN {X 8.954, Y 14.467, Z 5.950} C_DIS
   LIN {X 8.915, Y 15.169, Z 5.950} C_DIS
   LIN {X 8.896, Y 15.460, Z 5.950} C_DIS
   LIN {X 8.850, Y 16.154, Z 5.950} C_DIS
   LIN {X 8.776, Y 17.103, Z 5.950} C_DIS
   LIN {X 8.723, Y 17.799, Z 5.950} C_DIS
   LIN {X 8.660, Y 18.488, Z 5.950} C_DIS
   LIN {X 8.575, Y 19.398, Z 5.950} C_DIS
   LIN {X 8.504, Y 20.102, Z 5.950} C_DIS
   LIN {X 8.406, Y 20.942, Z 5.950} C_DIS
   LIN {X 8.333, Y 21.600, Z 5.950} C_DIS
   LIN {X 8.254, Y 22.252, Z 5.950} C_DIS
   LIN {X 8.203, Y 22.641, Z 5.950} C_DIS
   LIN {X 8.126, Y 23.237, Z 5.950} C_DIS
   LIN {X 8.073, Y 23.612, Z 5.950} C_DIS
   LIN {X 7.988, Y 24.227, Z 5.950} C_DIS
   LIN {X 7.898, Y 24.835, Z 5.950} C_DIS
   LIN {X 7.804, Y 25.438, Z 5.950} C_DIS
   LIN {X 7.655, Y 26.384, Z 5.950} C_DIS
   LIN {X 7.545, Y 27.050, Z 5.950} C_DIS
   LIN {X 7.490, Y 27.362, Z 5.950} C_DIS
   LIN {X 7.376, Y 28.018, Z 5.950} C_DIS
   LIN {X 7.320, Y 28.323, Z 5.950} C_DIS
   LIN {X 7.202, Y 28.963, Z 5.950} C_DIS
   LIN {X 7.140, Y 29.284, Z 5.950} C_DIS
   LIN {X 7.011, Y 29.952, Z 5.950} C_DIS
   LIN {X 6.946, Y 30.275, Z 5.950} C_DIS
   LIN {X 6.808, Y 30.955, Z 5.950} C_DIS
   LIN {X 6.738, Y 31.286, Z 5.950} C_DIS
   LIN {X 6.598, Y 31.943, Z 5.950} C_DIS
   LIN {X 6.491, Y 32.421, Z 5.950} C_DIS
   LIN {X 6.185, Y 33.702, Z 5.950} C_DIS
   LIN {X 5.763, Y 35.513, Z 5.950} C_DIS
   LIN {X 5.441, Y 36.745, Z 5.950} C_DIS
   LIN {X 5.296, Y 37.297, Z 5.950} C_DIS
   LIN {X 5.120, Y 37.933, Z 5.950} C_DIS
   LIN {X 4.900, Y 38.730, Z 5.950} C_DIS
   LIN {X 4.636, Y 39.267, Z 5.950} C_DIS
   LIN {X 4.250, Y 40.051, Z 5.950} C_DIS
   LIN {X 3.168, Y 40.984, Z 5.950} C_DIS
   LIN {X 2.966, Y 41.165, Z 5.950} C_DIS
   LIN {X 2.852, Y 41.218, Z 5.950} C_DIS
   LIN {X 1.303, Y 41.654, Z 5.950} C_DIS
   LIN {X 1.094, Y 41.651, Z 5.950} C_DIS
   LIN {X -0.822, Y 41.203, Z 5.950} C_DIS
   LIN {X -1.173, Y 40.979, Z 5.950} C_DIS
   LIN {X -1.649, Y 40.450, Z 5.950} C_DIS
   LIN {X -2.357, Y 39.755, Z 5.950} C_DIS
   LIN {X -2.626, Y 39.060, Z 5.950} C_DIS
   LIN {X -2.886, Y 38.271, Z 5.950} C_DIS
   LIN {X -2.833, Y 37.112, Z 5.950} C_DIS
   LIN {X -2.824, Y 36.808, Z 5.950} C_DIS
   LIN {X -2.792, Y 36.657, Z 5.950} C_DIS
   LIN {X -2.567, Y 35.583, Z 5.950} C_DIS
   LIN {X -2.333, Y 34.393, Z 5.950} C_DIS
   LIN {X -2.285, Y 34.154, Z 5.950} C_DIS
   LIN {X -2.223, Y 33.807, Z 5.950} C_DIS
   LIN {X -2.043, Y 32.704, Z 5.950} C_DIS
   LIN {X -1.832, Y 31.449, Z 5.950} C_DIS
   LIN {X -1.797, Y 31.217, Z 5.950} C_DIS
   LIN {X -1.680, Y 30.374, Z 5.950} C_DIS
   LIN {X -1.579, Y 29.568, Z 5.950} C_DIS
   LIN {X -1.537, Y 29.235, Z 5.950} C_DIS
   LIN {X -1.448, Y 28.433, Z 5.950} C_DIS
   LIN {X -1.394, Y 27.855, Z 5.950} C_DIS
   LIN {X -1.315, Y 27.045, Z 5.950} C_DIS
   LIN {X -1.248, Y 26.244, Z 5.950} C_DIS
   LIN {X -1.193, Y 25.446, Z 5.950} C_DIS
   LIN {X -1.180, Y 25.248, Z 5.950} C_DIS
   LIN {X -1.135, Y 24.451, Z 5.950} C_DIS
   LIN {X -1.101, Y 23.647, Z 5.950} C_DIS
   LIN {X -1.083, Y 23.242, Z 5.950} C_DIS
   LIN {X -1.060, Y 22.449, Z 5.950} C_DIS
   LIN {X -1.055, Y 22.245, Z 5.950} C_DIS
   LIN {X -1.043, Y 21.449, Z 5.950} C_DIS
   LIN {X -1.041, Y 21.242, Z 5.950} C_DIS
   LIN {X -1.040, Y 20.452, Z 5.950} C_DIS
   LIN {X -1.042, Y 20.139, Z 5.950} C_DIS
   LIN {X -1.072, Y 18.568, Z 5.950} C_DIS
   LIN {X -1.080, Y 18.251, Z 5.950} C_DIS
   LIN {X -1.112, Y 17.461, Z 5.950} C_DIS
   LIN {X -1.121, Y 17.244, Z 5.950} C_DIS
   LIN {X -1.162, Y 16.476, Z 5.950} C_DIS
   LIN {X -1.174, Y 16.261, Z 5.950} C_DIS
   LIN {X -1.224, Y 15.526, Z 5.950} C_DIS
   LIN {X -1.235, Y 15.356, Z 5.950} C_DIS
   LIN {X -1.296, Y 14.586, Z 5.950} C_DIS
   LIN {X -1.307, Y 14.452, Z 5.950} C_DIS
   LIN {X -1.387, Y 13.597, Z 5.950} C_DIS
   LIN {X -1.481, Y 12.712, Z 5.950} C_DIS
   LIN {X -1.592, Y 11.781, Z 5.950} C_DIS
   LIN {X -1.624, Y 11.492, Z 5.950} C_DIS
   LIN {X -1.768, Y 10.428, Z 5.950} C_DIS
   LIN {X -1.921, Y 9.405, Z 5.950} C_DIS
   LIN {X -2.083, Y 8.420, Z 5.950} C_DIS
   LIN {X -2.103, Y 8.308, Z 5.950} C_DIS
   LIN {X -2.264, Y 7.407, Z 5.950} C_DIS
   LIN {X -2.328, Y 7.077, Z 5.950} C_DIS
   LIN {X -2.477, Y 6.310, Z 5.950} C_DIS
   LIN {X -2.597, Y 5.735, Z 5.950} C_DIS
   LIN {X -2.683, Y 5.328, Z 5.950} C_DIS
   LIN {X -2.855, Y 4.560, Z 5.950} C_DIS
   LIN {X -2.906, Y 4.336, Z 5.950} C_DIS
   LIN {X -3.087, Y 3.577, Z 5.950} C_DIS
   LIN {X -3.141, Y 3.353, Z 5.950} C_DIS
   LIN {X -3.559, Y 1.741, Z 5.950} C_DIS
   LIN {X -3.593, Y 1.614, Z 5.950} C_DIS
   LIN {X -4.119, Y -0.201, Z 5.950} C_DIS
   LIN {X -4.322, Y -0.881, Z 5.950} C_DIS
   LIN {X -4.698, Y -2.043, Z 5.950} C_DIS
   LIN {X -4.829, Y -2.444, Z 5.950} C_DIS
   LIN {X -5.071, Y -3.148, Z 5.950} C_DIS
   LIN {X -5.156, Y -3.394, Z 5.950} C_DIS
   LIN {X -5.402, Y -4.078, Z 5.950} C_DIS
   LIN {X -5.490, Y -4.320, Z 5.950} C_DIS
   LIN {X -5.746, Y -5.003, Z 5.950} C_DIS
   LIN {X -5.840, Y -5.253, Z 5.950} C_DIS
   LIN {X -6.109, Y -5.941, Z 5.950} C_DIS
   LIN {X -6.207, Y -6.191, Z 5.950} C_DIS
   LIN {X -6.490, Y -6.886, Z 5.950} C_DIS
   LIN {X -6.773, Y -7.556, Z 5.950} C_DIS
   LIN {X -7.066, Y -8.224, Z 5.950} C_DIS
   LIN {X -7.364, Y -8.876, Z 5.950} C_DIS
   LIN {X -7.593, Y -9.409, Z 5.950} C_DIS
   LIN {X -7.839, Y -9.964, Z 5.950} C_DIS
   LIN {X -8.224, Y -10.777, Z 5.950} C_DIS
   LIN {X -8.614, Y -11.575, Z 5.950} C_DIS
   LIN {X -9.021, Y -12.378, Z 5.950} C_DIS
   LIN {X -9.603, Y -13.478, Z 5.950} C_DIS
   LIN {X -10.184, Y -14.561, Z 5.950} C_DIS
   LIN {X -11.528, Y -16.870, Z 5.950} C_DIS
   LIN {X -11.582, Y -16.964, Z 5.950} C_DIS
   LIN {X -12.697, Y -18.736, Z 5.950} C_DIS
   LIN {X -13.450, Y -20.263, Z 5.950} C_DIS
   LIN {X -13.539, Y -20.419, Z 5.950} C_DIS
   LIN {X -13.638, Y -20.658, Z 5.950} C_DIS
   LIN {X -13.671, Y -20.983, Z 5.950} C_DIS
   LIN {X -14.135, Y -24.189, Z 5.950} C_DIS
   LIN {X -14.097, Y -24.568, Z 5.950} C_DIS
   LIN {X -13.999, Y -25.075, Z 5.950} C_DIS
   LIN {X -13.838, Y -25.989, Z 5.950} C_DIS
   LIN {X -13.659, Y -26.578, Z 5.950} C_DIS
   LIN {X -13.248, Y -27.486, Z 5.950} C_DIS
   LIN {X -13.065, Y -27.917, Z 5.950} C_DIS
   LIN {X -12.825, Y -28.347, Z 5.950} C_DIS
   LIN {X -12.553, Y -28.730, Z 5.950} C_DIS
   LIN {X -12.117, Y -29.337, Z 5.950} C_DIS
   LIN {X -11.718, Y -29.788, Z 5.950} C_DIS
   LIN {X -10.671, Y -30.574, Z 5.950} C_DIS
   LIN {X -10.221, Y -30.988, Z 5.950} C_DIS
   LIN {X -9.741, Y -31.343, Z 5.950} C_DIS
   LIN {X -9.221, Y -31.649, Z 5.950} C_DIS
   LIN {X -8.642, Y -31.910, Z 5.950} C_DIS
   LIN {X -8.046, Y -32.106, Z 5.950} C_DIS
   LIN {X -7.423, Y -32.241, Z 5.950} C_DIS
   LIN {X -6.526, Y -32.500, Z 5.950} C_DIS
   LIN {X -5.934, Y -32.563, Z 5.950} C_DIS
   LIN {X -5.115, Y -32.556, Z 5.950} C_DIS
   LIN {X -4.433, Y -32.557, Z 5.950} C_DIS
   LIN {X -3.739, Y -32.481, Z 5.950} C_DIS
   LIN {X -3.034, Y -32.329, Z 5.950} C_DIS
   LIN {X -2.323, Y -32.093, Z 5.950} C_DIS
   LIN {X -1.629, Y -31.779, Z 5.950} C_DIS
   LIN {X -0.964, Y -31.549, Z 5.950} C_DIS
   LIN {X -0.200, Y -31.037, Z 5.950} C_DIS
   LIN {X 0.448, Y -30.622, Z 5.950} C_DIS
   LIN {X 0.720, Y -30.396, Z 5.950} C_DIS
   LIN {X 0.877, Y -30.225, Z 5.950} C_DIS
   LIN {X 2.457, Y -28.372, Z 5.950} C_DIS
   LIN {X 2.639, Y -28.101, Z 5.950} C_DIS
   LIN {X 2.813, Y -27.711, Z 5.950} C_DIS
   LIN {X 3.417, Y -26.398, Z 5.950} C_DIS
   LIN {X 4.015, Y -24.554, Z 5.950} C_DIS
   LIN {X 4.560, Y -22.762, Z 5.950} C_DIS
   LIN {X 4.905, Y -21.595, Z 5.950} C_DIS
   LIN {X 5.034, Y -21.112, Z 5.950} C_DIS
   LIN {X 5.191, Y -20.497, Z 5.950} C_DIS
   LIN {X 5.502, Y -19.406, Z 5.950} C_DIS
   LIN {X 5.533, Y -19.295, Z 5.950} C_DIS
   LIN {X 5.562, Y -19.188, Z 5.950} C_DIS
   LIN {X 5.784, Y -18.319, Z 5.950} C_DIS
   LIN {X 5.819, Y -18.185, Z 5.950} C_DIS
   LIN {X 5.849, Y -18.065, Z 5.950} C_DIS
   LIN {X 6.123, Y -16.940, Z 5.950} C_DIS
   LIN {X 6.432, Y -15.610, Z 5.950} C_DIS
   LIN {X 6.648, Y -14.631, Z 5.950} C_DIS
   LIN {X 6.853, Y -13.656, Z 5.950} C_DIS
   LIN {X 6.895, Y -13.442, Z 5.950} C_DIS
   LIN {X 7.079, Y -12.531, Z 5.950} C_DIS
   LIN {X 7.246, Y -11.659, Z 5.950} C_DIS
   LIN {X 7.322, Y -11.236, Z 5.950} C_DIS
   LIN {X 7.611, Y -9.598, Z 5.950} C_DIS
   LIN {X 7.717, Y -8.895, Z 5.950} C_DIS
   LIN {X 7.812, Y -8.330, Z 5.950} C_DIS
   LIN {X 7.938, Y -7.518, Z 5.950} C_DIS
   LIN {X 8.068, Y -6.618, Z 5.950} C_DIS
   LIN {X 8.199, Y -5.649, Z 5.950} C_DIS
   LIN {X 8.324, Y -4.652, Z 5.950} C_DIS
   LIN {X 8.440, Y -3.658, Z 5.950} C_DIS
   LIN {X 8.453, Y -3.528, Z 5.950} C_DIS
   LIN {X 8.587, Y -2.262, Z 5.950} C_DIS
   LIN {X 8.650, Y -1.572, Z 5.950} C_DIS
   LIN {X 8.732, Y -0.670, Z 5.950} C_DIS
   LIN {X 8.790, Y 0.232, Z 5.950} C_DIS
   LIN {X 8.851, Y 0.980, Z 5.950} C_DIS
   LIN {X 8.904, Y 1.725, Z 5.950} C_DIS
   LIN {X 8.950, Y 2.472, Z 5.950} C_DIS
   LIN {X 8.990, Y 3.223, Z 5.950} C_DIS
   LIN {X 9.022, Y 3.950, Z 5.950} C_DIS
   LIN {X 9.043, Y 4.479, Z 5.950} C_DIS
   LIN {X 9.068, Y 5.196, Z 5.950} C_DIS
   LIN {X 9.074, Y 5.455, Z 5.950} C_DIS
   LIN {X 9.093, Y 6.182, Z 5.950} C_DIS
   LIN {X 9.098, Y 6.456, Z 5.950} C_DIS
   LIN {X 9.110, Y 7.202, Z 5.950} C_DIS
   LIN {X 9.112, Y 7.470, Z 5.950} C_DIS
   LIN {X 9.117, Y 8.225, Z 5.950} C_DIS
   LIN {X 9.115, Y 8.954, Z 5.950} C_DIS
   LIN {X 9.112, Y 9.511, Z 5.950} C_DIS
   LIN {X 9.104, Y 10.199, Z 5.950} C_DIS
   LIN {X 9.099, Y 10.465, Z 5.950} C_DIS
   LIN {X 9.085, Y 11.172, Z 5.950} C_DIS
   LIN {X 9.077, Y 11.448, Z 5.950} C_DIS
   LIN {X 9.056, Y 12.181, Z 5.950} C_DIS
   LIN {X 9.045, Y 12.470, Z 5.950} C_DIS
   LIN {X 9.017, Y 13.187, Z 5.950}
   LaserEnd_Ext()
   LIN {X -12.280, Y -20.151, Z 5.950}
   LaserStart_Ext()
   LIN {X -12.280, Y -27.208, Z 5.950}
   LaserEnd_Ext()
   LIN {X -11.280, Y -28.774, Z 5.950}
   LaserStart_Ext()
   LIN {X -11.280, Y -18.361, Z 5.950}
   LaserEnd_Ext()
   LIN {X -10.280, Y -16.714, Z 5.950}
   LaserStart_Ext()
   LIN {X -10.280, Y -29.618, Z 5.950}
   LaserEnd_Ext()
   LIN {X -9.280, Y -30.440, Z 5.950}
   LaserStart_Ext()
   LIN {X -9.280, Y -14.990, Z 5.950}
   LaserEnd_Ext()
   LIN {X -8.280, Y -13.116, Z 5.950}
   LaserStart_Ext()
   LIN {X -8.280, Y -30.977, Z 5.950}
   LaserEnd_Ext()
   LIN {X -7.280, Y -31.249, Z 5.950}
   LaserStart_Ext()
   LIN {X -7.280, Y -11.121, Z 5.950}
   LaserEnd_Ext()
   LIN {X -6.280, Y -8.910, Z 5.950}
   LaserStart_Ext()
   LIN {X -6.280, Y -31.520, Z 5.950}
   LaserEnd_Ext()
   LIN {X -5.280, Y -31.558, Z 5.950}
   LaserStart_Ext()
   LIN {X -5.280, Y -6.566, Z 5.950}
   LaserEnd_Ext()
   LIN {X -4.280, Y -3.912, Z 5.950}
   LaserStart_Ext()
   LIN {X -4.280, Y -31.534, Z 5.950}
   LaserEnd_Ext()
   LIN {X -3.280, Y -31.357, Z 5.950}
   LaserStart_Ext()
   LIN {X -3.280, Y -0.886, Z 5.950}
   LaserEnd_Ext()
   LIN {X -2.280, Y 2.689, Z 5.950}
   LaserStart_Ext()
   LIN {X -2.280, Y -30.976, Z 5.950}
   LaserEnd_Ext()
   LIN {X -1.280, Y -30.557, Z 5.950}
   LaserStart_Ext()
   LIN {X -1.280, Y 7.230, Z 5.950}
   LaserEnd_Ext()
   LIN {X -1.280, Y 34.213, Z 5.950}
   LaserStart_Ext()
   LIN {X -1.280, Y 39.411, Z 5.950}
   LaserEnd_Ext()
   LIN {X -0.280, Y 40.303, Z 5.950}
   LaserStart_Ext()
   LIN {X -0.280, Y 26.664, Z 5.950}
   LaserEnd_Ext()
   LIN {X -0.280, Y 14.756, Z 5.950}
   LaserStart_Ext()
   LIN {X -0.280, Y -29.901, Z 5.950}
   LaserEnd_Ext()
   LIN {X 0.720, Y -28.868, Z 5.950}
   LaserStart_Ext()
   LIN {X 0.720, Y 40.537, Z 5.950}
   LaserEnd_Ext()
   LIN {X 1.720, Y 40.497, Z 5.950}
   LaserStart_Ext()
   LIN {X 1.720, Y -27.675, Z 5.950}
   LaserEnd_Ext()
   LIN {X 2.720, Y -25.306, Z 5.950}
   LaserStart_Ext()
   LIN {X 2.720, Y 40.049, Z 5.950}
   LaserEnd_Ext()
   LIN {X 3.720, Y 38.864, Z 5.950}
   LaserStart_Ext()
   LIN {X 3.720, Y -22.076, Z 5.950}
   LaserEnd_Ext()
   LIN {X 4.720, Y -18.444, Z 5.950}
   LaserStart_Ext()
   LIN {X 4.720, Y 35.548, Z 5.950}
   LaserEnd_Ext()
   LIN {X 5.720, Y 31.263, Z 5.950}
   LaserStart_Ext()
   LIN {X 5.720, Y -14.183, Z 5.950}
   LaserEnd_Ext()
   LIN {X 6.720, Y -8.797, Z 5.950}
   LaserStart_Ext()
   LIN {X 6.720, Y 25.893, Z 5.950}
   LaserEnd_Ext()
   LIN {X 7.720, Y 17.785, Z 5.950}
   LaserStart_Ext()
   LIN {X 7.720, Y -0.756, Z 5.950}
   LaserEnd_Ext()
   LIN {X -2.449, Y 6.507, Z 6.800}
   LaserStart_Ext()
   LIN {X -2.518, Y 6.147, Z 6.800} C_DIS
   LIN {X -2.561, Y 5.946, Z 6.800} C_DIS
   LIN {X -2.736, Y 5.114, Z 6.800} C_DIS
   LIN {X -2.818, Y 4.748, Z 6.800} C_DIS
   LIN {X -2.959, Y 4.122, Z 6.800} C_DIS
   LIN {X -3.046, Y 3.761, Z 6.800} C_DIS
   LIN {X -3.196, Y 3.139, Z 6.800} C_DIS
   LIN {X -3.394, Y 2.375, Z 6.800} C_DIS
   LIN {X -3.719, Y 1.152, Z 6.800} C_DIS
   LIN {X -3.943, Y 0.379, Z 6.800} C_DIS
   LIN {X -4.401, Y -1.152, Z 6.800} C_DIS
   LIN {X -4.539, Y -1.579, Z 6.800} C_DIS
   LIN {X -4.892, Y -2.658, Z 6.800} C_DIS
   LIN {X -4.991, Y -2.947, Z 6.800} C_DIS
   LIN {X -5.219, Y -3.605, Z 6.800} C_DIS
   LIN {X -5.319, Y -3.884, Z 6.800} C_DIS
   LIN {X -5.554, Y -4.531, Z 6.800} C_DIS
   LIN {X -5.658, Y -4.809, Z 6.800} C_DIS
   LIN {X -5.908, Y -5.471, Z 6.800} C_DIS
   LIN {X -6.016, Y -5.749, Z 6.800} C_DIS
   LIN {X -6.276, Y -6.408, Z 6.800} C_DIS
   LIN {X -6.389, Y -6.688, Z 6.800} C_DIS
   LIN {X -6.503, Y -6.958, Z 6.800} C_DIS
   LIN {X -6.622, Y -7.227, Z 6.800} C_DIS
   LIN {X -6.742, Y -7.490, Z 6.800} C_DIS
   LIN {X -7.335, Y -8.869, Z 6.800} C_DIS
   LIN {X -7.974, Y -10.307, Z 6.800} C_DIS
   LIN {X -8.286, Y -10.968, Z 6.800} C_DIS
   LIN {X -8.604, Y -11.617, Z 6.800} C_DIS
   LIN {X -8.935, Y -12.269, Z 6.800} C_DIS
   LIN {X -10.029, Y -14.338, Z 6.800} C_DIS
   LIN {X -10.222, Y -14.700, Z 6.800} C_DIS
   LIN {X -11.365, Y -16.671, Z 6.800} C_DIS
   LIN {X -12.238, Y -18.091, Z 6.800} C_DIS
   LIN {X -12.630, Y -18.714, Z 6.800} C_DIS
   LIN {X -13.036, Y -19.537, Z 6.800} C_DIS
   LIN {X -13.604, Y -20.781, Z 6.800} C_DIS
   LIN {X -14.011, Y -23.754, Z 6.800} C_DIS
   LIN {X -14.059, Y -24.085, Z 6.800} C_DIS
   LIN {X -13.693, Y -26.180, Z 6.800} C_DIS
   LIN {X -13.638, Y -26.361, Z 6.800} C_DIS
   LIN {X -13.059, Y -27.640, Z 6.800} C_DIS
   LIN {X -12.833, Y -28.157, Z 6.800} C_DIS
   LIN {X -12.754, Y -28.271, Z 6.800} C_DIS
   LIN {X -12.537, Y -28.574, Z 6.800} C_DIS
   LIN {X -11.914, Y -29.441, Z 6.800} C_DIS
   LIN {X -11.790, Y -29.582, Z 6.800} C_DIS
   LIN {X -9.462, Y -31.332, Z 6.800} C_DIS
   LIN {X -9.316, Y -31.466, Z 6.800} C_DIS
   LIN {X -9.161, Y -31.581, Z 6.800} C_DIS
   LIN {X -8.992, Y -31.680, Z 6.800} C_DIS
   LIN {X -8.804, Y -31.765, Z 6.800} C_DIS
   LIN {X -8.611, Y -31.829, Z 6.800} C_DIS
   LIN {X -8.409, Y -31.872, Z 6.800} C_DIS
   LIN {X -6.305, Y -32.479, Z 6.800} C_DIS
   LIN {X -4.299, Y -32.471, Z 6.800} C_DIS
   LIN {X -3.965, Y -32.471, Z 6.800} C_DIS
   LIN {X -3.626, Y -32.434, Z 6.800} C_DIS
   LIN {X -3.282, Y -32.360, Z 6.800} C_DIS
   LIN {X -2.934, Y -32.245, Z 6.800} C_DIS
   LIN {X -2.595, Y -32.091, Z 6.800} C_DIS
   LIN {X -0.843, Y -31.485, Z 6.800} C_DIS
   LIN {X 0.468, Y -30.607, Z 6.800} C_DIS
   LIN {X 0.774, Y -30.370, Z 6.800} C_DIS
   LIN {X 2.549, Y -28.303, Z 6.800} C_DIS
   LIN {X 3.010, Y -27.410, Z 6.800} C_DIS
   LIN {X 3.504, Y -26.336, Z 6.800} C_DIS
   LIN {X 3.777, Y -25.496, Z 6.800} C_DIS
   LIN {X 4.100, Y -24.477, Z 6.800} C_DIS
   LIN {X 4.447, Y -23.319, Z 6.800} C_DIS
   LIN {X 4.712, Y -22.445, Z 6.800} C_DIS
   LIN {X 4.881, Y -21.874, Z 6.800} C_DIS
   LIN {X 5.271, Y -20.418, Z 6.800} C_DIS
   LIN {X 5.743, Y -18.563, Z 6.800} C_DIS
   LIN {X 5.910, Y -17.977, Z 6.800} C_DIS
   LIN {X 6.028, Y -17.514, Z 6.800} C_DIS
   LIN {X 6.172, Y -16.924, Z 6.800} C_DIS
   LIN {X 6.314, Y -16.312, Z 6.800} C_DIS
   LIN {X 6.542, Y -15.298, Z 6.800} C_DIS
   LIN {X 6.658, Y -14.772, Z 6.800} C_DIS
   LIN {X 6.763, Y -14.271, Z 6.800} C_DIS
   LIN {X 6.863, Y -13.797, Z 6.800} C_DIS
   LIN {X 7.073, Y -12.726, Z 6.800} C_DIS
   LIN {X 7.154, Y -12.325, Z 6.800} C_DIS
   LIN {X 7.228, Y -11.941, Z 6.800} C_DIS
   LIN {X 7.467, Y -10.602, Z 6.800} C_DIS
   LIN {X 7.594, Y -9.881, Z 6.800} C_DIS
   LIN {X 7.928, Y -7.650, Z 6.800} C_DIS
   LIN {X 7.981, Y -7.339, Z 6.800} C_DIS
   LIN {X 8.050, Y -6.893, Z 6.800} C_DIS
   LIN {X 8.122, Y -6.398, Z 6.800} C_DIS
   LIN {X 8.193, Y -5.865, Z 6.800} C_DIS
   LIN {X 8.251, Y -5.406, Z 6.800} C_DIS
   LIN {X 8.318, Y -4.870, Z 6.800} C_DIS
   LIN {X 8.418, Y -4.011, Z 6.800} C_DIS
   LIN {X 8.449, Y -3.745, Z 6.800} C_DIS
   LIN {X 8.512, Y -3.140, Z 6.800} C_DIS
   LIN {X 8.579, Y -2.501, Z 6.800} C_DIS
   LIN {X 8.637, Y -1.857, Z 6.800} C_DIS
   LIN {X 8.747, Y -0.642, Z 6.800} C_DIS
   LIN {X 8.905, Y 1.800, Z 6.800} C_DIS
   LIN {X 8.930, Y 2.100, Z 6.800} C_DIS
   LIN {X 8.951, Y 2.400, Z 6.800} C_DIS
   LIN {X 8.970, Y 2.700, Z 6.800} C_DIS
   LIN {X 8.986, Y 3.002, Z 6.800} C_DIS
   LIN {X 8.998, Y 3.293, Z 6.800} C_DIS
   LIN {X 9.054, Y 4.688, Z 6.800} C_DIS
   LIN {X 9.064, Y 4.978, Z 6.800} C_DIS
   LIN {X 9.082, Y 5.665, Z 6.800} C_DIS
   LIN {X 9.089, Y 5.960, Z 6.800} C_DIS
   LIN {X 9.101, Y 6.692, Z 6.800} C_DIS
   LIN {X 9.106, Y 6.991, Z 6.800} C_DIS
   LIN {X 9.112, Y 7.706, Z 6.800} C_DIS
   LIN {X 9.114, Y 8.008, Z 6.800} C_DIS
   LIN {X 9.113, Y 8.299, Z 6.800} C_DIS
   LIN {X 9.104, Y 9.741, Z 6.800} C_DIS
   LIN {X 9.101, Y 10.009, Z 6.800} C_DIS
   LIN {X 9.087, Y 10.695, Z 6.800} C_DIS
   LIN {X 9.082, Y 10.969, Z 6.800} C_DIS
   LIN {X 9.061, Y 11.678, Z 6.800} C_DIS
   LIN {X 9.053, Y 11.961, Z 6.800} C_DIS
   LIN {X 9.025, Y 12.700, Z 6.800} C_DIS
   LIN {X 9.015, Y 12.976, Z 6.800} C_DIS
   LIN {X 8.981, Y 13.694, Z 6.800} C_DIS
   LIN {X 8.968, Y 13.965, Z 6.800} C_DIS
   LIN {X 8.928, Y 14.687, Z 6.800} C_DIS
   LIN {X 8.913, Y 14.952, Z 6.800} C_DIS
   LIN {X 8.866, Y 15.679, Z 6.800} C_DIS
   LIN {X 8.849, Y 15.940, Z 6.800} C_DIS
   LIN {X 8.767, Y 16.987, Z 6.800} C_DIS
   LIN {X 8.705, Y 17.777, Z 6.800} C_DIS
   LIN {X 8.641, Y 18.440, Z 6.800} C_DIS
   LIN {X 8.538, Y 19.547, Z 6.800} C_DIS
   LIN {X 8.506, Y 19.859, Z 6.800} C_DIS
   LIN {X 8.266, Y 21.919, Z 6.800} C_DIS
   LIN {X 8.248, Y 22.078, Z 6.800} C_DIS
   LIN {X 8.229, Y 22.235, Z 6.800} C_DIS
   LIN {X 8.105, Y 23.175, Z 6.800} C_DIS
   LIN {X 7.968, Y 24.145, Z 6.800} C_DIS
   LIN {X 7.949, Y 24.279, Z 6.800} C_DIS
   LIN {X 7.585, Y 26.600, Z 6.800} C_DIS
   LIN {X 7.546, Y 26.835, Z 6.800} C_DIS
   LIN {X 7.417, Y 27.574, Z 6.800} C_DIS
   LIN {X 7.377, Y 27.804, Z 6.800} C_DIS
   LIN {X 7.245, Y 28.522, Z 6.800} C_DIS
   LIN {X 7.204, Y 28.745, Z 6.800} C_DIS
   LIN {X 7.058, Y 29.502, Z 6.800} C_DIS
   LIN {X 7.013, Y 29.734, Z 6.800} C_DIS
   LIN {X 6.860, Y 30.492, Z 6.800} C_DIS
   LIN {X 6.813, Y 30.726, Z 6.800} C_DIS
   LIN {X 6.649, Y 31.502, Z 6.800} C_DIS
   LIN {X 6.601, Y 31.727, Z 6.800} C_DIS
   LIN {X 6.352, Y 32.836, Z 6.800} C_DIS
   LIN {X 5.776, Y 35.247, Z 6.800} C_DIS
   LIN {X 5.712, Y 35.510, Z 6.800} C_DIS
   LIN {X 5.621, Y 35.853, Z 6.800} C_DIS
   LIN {X 5.225, Y 37.365, Z 6.800} C_DIS
   LIN {X 5.010, Y 38.139, Z 6.800} C_DIS
   LIN {X 4.825, Y 38.797, Z 6.800} C_DIS
   LIN {X 4.434, Y 39.583, Z 6.800} C_DIS
   LIN {X 4.171, Y 40.116, Z 6.800} C_DIS
   LIN {X 3.772, Y 40.460, Z 6.800} C_DIS
   LIN {X 2.850, Y 41.252, Z 6.800} C_DIS
   LIN {X 1.847, Y 41.531, Z 6.800} C_DIS
   LIN {X 1.156, Y 41.721, Z 6.800} C_DIS
   LIN {X 0.444, Y 41.513, Z 6.800} C_DIS
   LIN {X -1.108, Y 41.141, Z 6.800} C_DIS
   LIN {X -1.647, Y 40.610, Z 6.800} C_DIS
   LIN {X -2.384, Y 39.888, Z 6.800} C_DIS
   LIN {X -2.723, Y 39.011, Z 6.800} C_DIS
   LIN {X -2.949, Y 38.406, Z 6.800} C_DIS
   LIN {X -2.930, Y 38.076, Z 6.800} C_DIS
   LIN {X -2.894, Y 36.857, Z 6.800} C_DIS
   LIN {X -2.671, Y 35.803, Z 6.800} C_DIS
   LIN {X -2.636, Y 35.632, Z 6.800} C_DIS
   LIN {X -2.571, Y 35.304, Z 6.800} C_DIS
   LIN {X -2.323, Y 34.061, Z 6.800} C_DIS
   LIN {X -2.105, Y 32.810, Z 6.800} C_DIS
   LIN {X -1.951, Y 31.889, Z 6.800} C_DIS
   LIN {X -1.800, Y 30.888, Z 6.800} C_DIS
   LIN {X -1.744, Y 30.488, Z 6.800} C_DIS
   LIN {X -1.697, Y 30.106, Z 6.800} C_DIS
   LIN {X -1.557, Y 29.008, Z 6.800} C_DIS
   LIN {X -1.517, Y 28.641, Z 6.800} C_DIS
   LIN {X -1.339, Y 26.751, Z 6.800} C_DIS
   LIN {X -1.304, Y 26.383, Z 6.800} C_DIS
   LIN {X -1.273, Y 26.020, Z 6.800} C_DIS
   LIN {X -1.248, Y 25.658, Z 6.800} C_DIS
   LIN {X -1.206, Y 25.024, Z 6.800} C_DIS
   LIN {X -1.186, Y 24.663, Z 6.800} C_DIS
   LIN {X -1.171, Y 24.299, Z 6.800} C_DIS
   LIN {X -1.112, Y 23.020, Z 6.800} C_DIS
   LIN {X -1.102, Y 22.663, Z 6.800} C_DIS
   LIN {X -1.086, Y 22.022, Z 6.800} C_DIS
   LIN {X -1.081, Y 21.665, Z 6.800} C_DIS
   LIN {X -1.073, Y 21.019, Z 6.800} C_DIS
   LIN {X -1.073, Y 20.666, Z 6.800} C_DIS
   LIN {X -1.078, Y 19.699, Z 6.800} C_DIS
   LIN {X -1.092, Y 18.999, Z 6.800} C_DIS
   LIN {X -1.117, Y 18.034, Z 6.800} C_DIS
   LIN {X -1.130, Y 17.684, Z 6.800} C_DIS
   LIN {X -1.159, Y 17.027, Z 6.800} C_DIS
   LIN {X -1.177, Y 16.688, Z 6.800} C_DIS
   LIN {X -1.214, Y 16.040, Z 6.800} C_DIS
   LIN {X -1.235, Y 15.716, Z 6.800} C_DIS
   LIN {X -1.276, Y 15.135, Z 6.800} C_DIS
   LIN {X -1.304, Y 14.777, Z 6.800} C_DIS
   LIN {X -1.349, Y 14.231, Z 6.800} C_DIS
   LIN {X -1.388, Y 13.813, Z 6.800} C_DIS
   LIN {X -1.434, Y 13.380, Z 6.800} C_DIS
   LIN {X -1.488, Y 12.925, Z 6.800} C_DIS
   LIN {X -1.667, Y 11.286, Z 6.800} C_DIS
   LIN {X -1.743, Y 10.728, Z 6.800} C_DIS
   LIN {X -1.825, Y 10.129, Z 6.800} C_DIS
   LIN {X -1.901, Y 9.624, Z 6.800} C_DIS
   LIN {X -1.987, Y 9.071, Z 6.800} C_DIS
   LIN {X -2.074, Y 8.545, Z 6.800} C_DIS
   LIN {X -2.219, Y 7.717, Z 6.800} C_DIS
   LIN {X -2.272, Y 7.418, Z 6.800} C_DIS
   LIN {X -2.449, Y 6.507, Z 6.800}
   LaserEnd_Ext()
   LIN {X -6.576, Y -31.360, Z 6.800}
   LaserStart_Ext()
   LIN {X -3.444, Y -31.360, Z 6.800}
   LaserEnd_Ext()
   LIN {X -0.961, Y -30.360, Z 6.800}
   LaserStart_Ext()
   LIN {X -9.091, Y -30.360, Z 6.800}
   LaserEnd_Ext()
   LIN {X -10.421, Y -29.360, Z 6.800}
   LaserStart_Ext()
   LIN {X 0.323, Y -29.360, Z 6.800}
   LaserEnd_Ext()
   LIN {X 1.182, Y -28.360, Z 6.800}
   LaserStart_Ext()
   LIN {X -11.460, Y -28.360, Z 6.800}
   LaserEnd_Ext()
   LIN {X -12.090, Y -27.360, Z 6.800}
   LaserStart_Ext()
   LIN {X 1.911, Y -27.360, Z 6.800}
   LaserEnd_Ext()
   LIN {X 2.392, Y -26.360, Z 6.800}
   LaserStart_Ext()
   LIN {X -12.541, Y -26.360, Z 6.800}
   LaserEnd_Ext()
   LIN {X -12.821, Y -25.360, Z 6.800}
   LaserStart_Ext()
   LIN {X 2.769, Y -25.360, Z 6.800}
   LaserEnd_Ext()
   LIN {X 3.088, Y -24.360, Z 6.800}
   LaserStart_Ext()
   LIN {X -12.997, Y -24.360, Z 6.800}
   LaserEnd_Ext()
   LIN {X -12.948, Y -23.360, Z 6.800}
   LaserStart_Ext()
   LIN {X 3.391, Y -23.360, Z 6.800}
   LaserEnd_Ext()
   LIN {X 3.693, Y -22.360, Z 6.800}
   LaserStart_Ext()
   LIN {X -12.811, Y -22.360, Z 6.800}
   LaserEnd_Ext()
   LIN {X -12.673, Y -21.360, Z 6.800}
   LaserStart_Ext()
   LIN {X 3.983, Y -21.360, Z 6.800}
   LaserEnd_Ext()
   LIN {X 4.251, Y -20.360, Z 6.800}
   LaserStart_Ext()
   LIN {X -12.312, Y -20.360, Z 6.800}
   LaserEnd_Ext()
   LIN {X -11.834, Y -19.360, Z 6.800}
   LaserStart_Ext()
   LIN {X 4.508, Y -19.360, Z 6.800}
   LaserEnd_Ext()
   LIN {X 4.762, Y -18.360, Z 6.800}
   LaserStart_Ext()
   LIN {X -11.230, Y -18.360, Z 6.800}
   LaserEnd_Ext()
   LIN {X -10.615, Y -17.360, Z 6.800}
   LaserStart_Ext()
   LIN {X 5.035, Y -17.360, Z 6.800}
   LaserEnd_Ext()
   LIN {X 5.276, Y -16.360, Z 6.800}
   LaserStart_Ext()
   LIN {X -10.029, Y -16.360, Z 6.800}
   LaserEnd_Ext()
   LIN {X -9.449, Y -15.360, Z 6.800}
   LaserStart_Ext()
   LIN {X 5.503, Y -15.360, Z 6.800}
   LaserEnd_Ext()
   LIN {X 5.722, Y -14.360, Z 6.800}
   LaserStart_Ext()
   LIN {X -8.910, Y -14.360, Z 6.800}
   LaserEnd_Ext()
   LIN {X -8.380, Y -13.360, Z 6.800}
   LaserStart_Ext()
   LIN {X 5.930, Y -13.360, Z 6.800}
   LaserEnd_Ext()
   LIN {X 6.127, Y -12.360, Z 6.800}
   LaserStart_Ext()
   LIN {X -7.859, Y -12.360, Z 6.800}
   LaserEnd_Ext()
   LIN {X -7.366, Y -11.360, Z 6.800}
   LaserStart_Ext()
   LIN {X 6.316, Y -11.360, Z 6.800}
   LaserEnd_Ext()
   LIN {X 6.494, Y -10.360, Z 6.800}
   LaserStart_Ext()
   LIN {X -6.903, Y -10.360, Z 6.800}
   LaserEnd_Ext()
   LIN {X -6.459, Y -9.360, Z 6.800}
   LaserStart_Ext()
   LIN {X 6.661, Y -9.360, Z 6.800}
   LaserEnd_Ext()
   LIN {X 6.811, Y -8.360, Z 6.800}
   LaserStart_Ext()
   LIN {X -6.027, Y -8.360, Z 6.800}
   LaserEnd_Ext()
   LIN {X -5.588, Y -7.360, Z 6.800}
   LaserStart_Ext()
   LIN {X 6.963, Y -7.360, Z 6.800}
   LaserEnd_Ext()
   LIN {X 7.117, Y -6.360, Z 6.800}
   LaserStart_Ext()
   LIN {X -5.182, Y -6.360, Z 6.800}
   LaserEnd_Ext()
   LIN {X -4.797, Y -5.360, Z 6.800}
   LaserStart_Ext()
   LIN {X 7.249, Y -5.360, Z 6.800}
   LaserEnd_Ext()
   LIN {X 7.371, Y -4.360, Z 6.800}
   LaserStart_Ext()
   LIN {X -4.428, Y -4.360, Z 6.800}
   LaserEnd_Ext()
   LIN {X -4.076, Y -3.360, Z 6.800}
   LaserStart_Ext()
   LIN {X 7.484, Y -3.360, Z 6.800}
   LaserEnd_Ext()
   LIN {X 7.588, Y -2.360, Z 6.800}
   LaserStart_Ext()
   LIN {X -3.742, Y -2.360, Z 6.800}
   LaserEnd_Ext()
   LIN {X -3.419, Y -1.360, Z 6.800}
   LaserStart_Ext()
   LIN {X 7.678, Y -1.360, Z 6.800}
   LaserEnd_Ext()
   LIN {X 7.764, Y -0.360, Z 6.800}
   LaserStart_Ext()
   LIN {X -3.120, Y -0.360, Z 6.800}
   LaserEnd_Ext()
   LIN {X -2.826, Y 0.640, Z 6.800}
   LaserStart_Ext()
   LIN {X 7.828, Y 0.640, Z 6.800}
   LaserEnd_Ext()
   LIN {X 7.893, Y 1.640, Z 6.800}
   LaserStart_Ext()
   LIN {X -2.555, Y 1.640, Z 6.800}
   LaserEnd_Ext()
   LIN {X -2.292, Y 2.640, Z 6.800}
   LaserStart_Ext()
   LIN {X 7.964, Y 2.640, Z 6.800}
   LaserEnd_Ext()
   LIN {X 8.011, Y 3.640, Z 6.800}
   LaserStart_Ext()
   LIN {X -2.046, Y 3.640, Z 6.800}
   LaserEnd_Ext()
   LIN {X -1.817, Y 4.640, Z 6.800}
   LaserStart_Ext()
   LIN {X 8.051, Y 4.640, Z 6.800}
   LaserEnd_Ext()
   LIN {X 8.081, Y 5.640, Z 6.800}
   LaserStart_Ext()
   LIN {X -1.603, Y 5.640, Z 6.800}
   LaserEnd_Ext()
   LIN {X -1.405, Y 6.640, Z 6.800}
   LaserStart_Ext()
   LIN {X 8.100, Y 6.640, Z 6.800}
   LaserEnd_Ext()
   LIN {X 8.111, Y 7.640, Z 6.800}
   LaserStart_Ext()
   LIN {X -1.217, Y 7.640, Z 6.800}
   LaserEnd_Ext()
   LIN {X -1.045, Y 8.640, Z 6.800}
   LaserStart_Ext()
   LIN {X 8.111, Y 8.640, Z 6.800}
   LaserEnd_Ext()
   LIN {X 8.105, Y 9.640, Z 6.800}
   LaserStart_Ext()
   LIN {X -0.888, Y 9.640, Z 6.800}
   LaserEnd_Ext()
   LIN {X -0.745, Y 10.640, Z 6.800}
   LaserStart_Ext()
   LIN {X 8.088, Y 10.640, Z 6.800}
   LaserEnd_Ext()
   LIN {X 8.062, Y 11.640, Z 6.800}
   LaserStart_Ext()
   LIN {X -0.622, Y 11.640, Z 6.800}
   LaserEnd_Ext()
   LIN {X -0.513, Y 12.640, Z 6.800}
   LaserStart_Ext()
   LIN {X 8.027, Y 12.640, Z 6.800}
   LaserEnd_Ext()
   LIN {X 7.982, Y 13.640, Z 6.800}
   LaserStart_Ext()
   LIN {X -0.400, Y 13.640, Z 6.800}
   LaserEnd_Ext()
   LIN {X -0.312, Y 14.640, Z 6.800}
   LaserStart_Ext()
   LIN {X 7.929, Y 14.640, Z 6.800}
   LaserEnd_Ext()
   LIN {X 7.866, Y 15.640, Z 6.800}
   LaserStart_Ext()
   LIN {X -0.238, Y 15.640, Z 6.800}
   LaserEnd_Ext()
   LIN {X -0.178, Y 16.640, Z 6.800}
   LaserStart_Ext()
   LIN {X 7.791, Y 16.640, Z 6.800}
   LaserEnd_Ext()
   LIN {X 7.713, Y 17.640, Z 6.800}
   LaserStart_Ext()
   LIN {X -0.131, Y 17.640, Z 6.800}
   LaserEnd_Ext()
   LIN {X -0.101, Y 18.640, Z 6.800}
   LaserStart_Ext()
   LIN {X 7.618, Y 18.640, Z 6.800}
   LaserEnd_Ext()
   LIN {X 7.523, Y 19.640, Z 6.800}
   LaserStart_Ext()
   LIN {X -0.079, Y 19.640, Z 6.800}
   LaserEnd_Ext()
   LIN {X -0.073, Y 20.640, Z 6.800}
   LaserStart_Ext()
   LIN {X 7.408, Y 20.640, Z 6.800}
   LaserEnd_Ext()
   LIN {X 7.291, Y 21.640, Z 6.800}
   LaserStart_Ext()
   LIN {X -0.080, Y 21.640, Z 6.800}
   LaserEnd_Ext()
   LIN {X -0.101, Y 22.640, Z 6.800}
   LaserStart_Ext()
   LIN {X 7.167, Y 22.640, Z 6.800}
   LaserEnd_Ext()
   LIN {X 7.030, Y 23.640, Z 6.800}
   LaserStart_Ext()
   LIN {X -0.140, Y 23.640, Z 6.800}
   LaserEnd_Ext()
   LIN {X -0.184, Y 24.640, Z 6.800}
   LaserStart_Ext()
   LIN {X 6.880, Y 24.640, Z 6.800}
   LaserEnd_Ext()
   LIN {X 6.723, Y 25.640, Z 6.800}
   LaserStart_Ext()
   LIN {X -0.245, Y 25.640, Z 6.800}
   LaserEnd_Ext()
   LIN {X -0.324, Y 26.640, Z 6.800}
   LaserStart_Ext()
   LIN {X 6.565, Y 26.640, Z 6.800}
   LaserEnd_Ext()
   LIN {X 6.390, Y 27.640, Z 6.800}
   LaserStart_Ext()
   LIN {X -0.418, Y 27.640, Z 6.800}
   LaserEnd_Ext()
   LIN {X -0.512, Y 28.640, Z 6.800}
   LaserStart_Ext()
   LIN {X 6.206, Y 28.640, Z 6.800}
   LaserEnd_Ext()
   LIN {X 6.012, Y 29.640, Z 6.800}
   LaserStart_Ext()
   LIN {X -0.629, Y 29.640, Z 6.800}
   LaserEnd_Ext()
   LIN {X -0.756, Y 30.640, Z 6.800}
   LaserStart_Ext()
   LIN {X 5.809, Y 30.640, Z 6.800}
   LaserEnd_Ext()
   LIN {X 5.596, Y 31.640, Z 6.800}
   LaserStart_Ext()
   LIN {X -0.902, Y 31.640, Z 6.800}
   LaserEnd_Ext()
   LIN {X -1.063, Y 32.640, Z 6.800}
   LaserStart_Ext()
   LIN {X 5.371, Y 32.640, Z 6.800}
   LaserEnd_Ext()
   LIN {X 5.132, Y 33.640, Z 6.800}
   LaserStart_Ext()
   LIN {X -1.235, Y 33.640, Z 6.800}
   LaserEnd_Ext()
   LIN {X -1.419, Y 34.640, Z 6.800}
   LaserStart_Ext()
   LIN {X 4.893, Y 34.640, Z 6.800}
   LaserEnd_Ext()
   LIN {X 4.643, Y 35.640, Z 6.800}
   LaserStart_Ext()
   LIN {X -1.618, Y 35.640, Z 6.800}
   LaserEnd_Ext()
   LIN {X -1.826, Y 36.640, Z 6.800}
   LaserStart_Ext()
   LIN {X 4.381, Y 36.640, Z 6.800}
   LaserEnd_Ext()
   LIN {X 4.110, Y 37.640, Z 6.800}
   LaserStart_Ext()
   LIN {X -1.917, Y 37.640, Z 6.800}
   LaserEnd_Ext()
   LIN {X -1.794, Y 38.640, Z 6.800}
   LaserStart_Ext()
   LIN {X 3.787, Y 38.640, Z 6.800}
   LaserEnd_Ext()
   LIN {X 3.193, Y 39.640, Z 6.800}
   LaserStart_Ext()
   LIN {X -1.208, Y 39.640, Z 6.800}
   LaserEnd_Ext()
   LIN {X 1.021, Y 40.640, Z 6.800}
   LaserStart_Ext()
   LIN {X 1.317, Y 40.640, Z 6.800}
   LaserEnd_Ext()
   LIN {X 6.579, Y 31.632, Z 7.650}
   LaserStart_Ext()
   LIN {X 6.744, Y 30.854, Z 7.650} C_DIS
   LIN {X 6.901, Y 30.069, Z 7.650} C_DIS
   LIN {X 7.074, Y 29.217, Z 7.650} C_DIS
   LIN {X 7.238, Y 28.360, Z 7.650} C_DIS
   LIN {X 7.388, Y 27.544, Z 7.650} C_DIS
   LIN {X 7.535, Y 26.701, Z 7.650} C_DIS
   LIN {X 7.579, Y 26.434, Z 7.650} C_DIS
   LIN {X 7.889, Y 24.481, Z 7.650} C_DIS
   LIN {X 8.041, Y 23.413, Z 7.650} C_DIS
   LIN {X 8.140, Y 22.712, Z 7.650} C_DIS
   LIN {X 8.231, Y 22.020, Z 7.650} C_DIS
   LIN {X 8.488, Y 19.798, Z 7.650} C_DIS
   LIN {X 8.506, Y 19.646, Z 7.650} C_DIS
   LIN {X 8.542, Y 19.273, Z 7.650} C_DIS
   LIN {X 8.691, Y 17.724, Z 7.650} C_DIS
   LIN {X 8.793, Y 16.422, Z 7.650} C_DIS
   LIN {X 8.847, Y 15.749, Z 7.650} C_DIS
   LIN {X 8.905, Y 14.857, Z 7.650} C_DIS
   LIN {X 8.955, Y 13.965, Z 7.650} C_DIS
   LIN {X 8.997, Y 13.067, Z 7.650} C_DIS
   LIN {X 9.013, Y 12.784, Z 7.650} C_DIS
   LIN {X 9.046, Y 11.895, Z 7.650} C_DIS
   LIN {X 9.071, Y 11.038, Z 7.650} C_DIS
   LIN {X 9.087, Y 10.203, Z 7.650} C_DIS
   LIN {X 9.099, Y 9.761, Z 7.650} C_DIS
   LIN {X 9.111, Y 7.989, Z 7.650} C_DIS
   LIN {X 9.111, Y 7.773, Z 7.650} C_DIS
   LIN {X 9.104, Y 6.857, Z 7.650} C_DIS
   LIN {X 9.088, Y 5.909, Z 7.650} C_DIS
   LIN {X 9.065, Y 5.024, Z 7.650} C_DIS
   LIN {X 9.058, Y 4.686, Z 7.650} C_DIS
   LIN {X 8.987, Y 2.895, Z 7.650} C_DIS
   LIN {X 8.978, Y 2.706, Z 7.650} C_DIS
   LIN {X 8.764, Y -0.598, Z 7.650} C_DIS
   LIN {X 8.578, Y -2.686, Z 7.650} C_DIS
   LIN {X 8.481, Y -3.611, Z 7.650} C_DIS
   LIN {X 8.349, Y -4.777, Z 7.650} C_DIS
   LIN {X 8.313, Y -5.089, Z 7.650} C_DIS
   LIN {X 8.188, Y -6.081, Z 7.650} C_DIS
   LIN {X 8.162, Y -6.268, Z 7.650} C_DIS
   LIN {X 8.140, Y -6.405, Z 7.650} C_DIS
   LIN {X 7.878, Y -8.158, Z 7.650} C_DIS
   LIN {X 7.604, Y -9.998, Z 7.650} C_DIS
   LIN {X 7.464, Y -10.768, Z 7.650} C_DIS
   LIN {X 7.154, Y -12.506, Z 7.650} C_DIS
   LIN {X 6.957, Y -13.507, Z 7.650} C_DIS
   LIN {X 6.872, Y -13.938, Z 7.650} C_DIS
   LIN {X 6.668, Y -14.913, Z 7.650} C_DIS
   LIN {X 6.413, Y -16.049, Z 7.650} C_DIS
   LIN {X 6.284, Y -16.620, Z 7.650} C_DIS
   LIN {X 6.181, Y -17.075, Z 7.650} C_DIS
   LIN {X 5.508, Y -19.723, Z 7.650} C_DIS
   LIN {X 4.887, Y -22.041, Z 7.650} C_DIS
   LIN {X 4.849, Y -22.179, Z 7.650} C_DIS
   LIN {X 4.180, Y -24.414, Z 7.650} C_DIS
   LIN {X 3.631, Y -26.144, Z 7.650} C_DIS
   LIN {X 3.590, Y -26.274, Z 7.650} C_DIS
   LIN {X 3.462, Y -26.497, Z 7.650} C_DIS
   LIN {X 2.374, Y -28.608, Z 7.650} C_DIS
   LIN {X 1.111, Y -30.078, Z 7.650} C_DIS
   LIN {X 0.009, Y -30.931, Z 7.650} C_DIS
   LIN {X -0.722, Y -31.421, Z 7.650} C_DIS
   LIN {X -3.418, Y -32.354, Z 7.650} C_DIS
   LIN {X -3.562, Y -32.388, Z 7.650} C_DIS
   LIN {X -6.216, Y -32.438, Z 7.650} C_DIS
   LIN {X -8.389, Y -31.806, Z 7.650} C_DIS
   LIN {X -9.153, Y -31.483, Z 7.650} C_DIS
   LIN {X -11.533, Y -29.696, Z 7.650} C_DIS
   LIN {X -11.716, Y -29.533, Z 7.650} C_DIS
   LIN {X -12.364, Y -28.625, Z 7.650} C_DIS
   LIN {X -12.877, Y -27.885, Z 7.650} C_DIS
   LIN {X -13.463, Y -26.548, Z 7.650} C_DIS
   LIN {X -13.667, Y -25.250, Z 7.650} C_DIS
   LIN {X -13.968, Y -24.183, Z 7.650} C_DIS
   LIN {X -13.921, Y -23.295, Z 7.650} C_DIS
   LIN {X -13.612, Y -21.044, Z 7.650} C_DIS
   LIN {X -12.777, Y -19.211, Z 7.650} C_DIS
   LIN {X -12.564, Y -18.691, Z 7.650} C_DIS
   LIN {X -12.199, Y -18.088, Z 7.650} C_DIS
   LIN {X -11.147, Y -16.378, Z 7.650} C_DIS
   LIN {X -10.454, Y -15.182, Z 7.650} C_DIS
   LIN {X -9.692, Y -13.754, Z 7.650} C_DIS
   LIN {X -8.848, Y -12.161, Z 7.650} C_DIS
   LIN {X -8.594, Y -11.658, Z 7.650} C_DIS
   LIN {X -8.349, Y -11.158, Z 7.650} C_DIS
   LIN {X -8.109, Y -10.649, Z 7.650} C_DIS
   LIN {X -7.077, Y -8.328, Z 7.650} C_DIS
   LIN {X -6.346, Y -6.631, Z 7.650} C_DIS
   LIN {X -6.179, Y -6.187, Z 7.650} C_DIS
   LIN {X -5.863, Y -5.386, Z 7.650} C_DIS
   LIN {X -5.557, Y -4.575, Z 7.650} C_DIS
   LIN {X -5.268, Y -3.777, Z 7.650} C_DIS
   LIN {X -5.061, Y -3.148, Z 7.650} C_DIS
   LIN {X -4.802, Y -2.401, Z 7.650} C_DIS
   LIN {X -4.402, Y -1.176, Z 7.650} C_DIS
   LIN {X -3.894, Y 0.529, Z 7.650} C_DIS
   LIN {X -3.790, Y 0.893, Z 7.650} C_DIS
   LIN {X -3.257, Y 2.902, Z 7.650} C_DIS
   LIN {X -3.012, Y 3.912, Z 7.650} C_DIS
   LIN {X -2.786, Y 4.909, Z 7.650} C_DIS
   LIN {X -2.539, Y 6.081, Z 7.650} C_DIS
   LIN {X -2.363, Y 6.991, Z 7.650} C_DIS
   LIN {X -2.291, Y 7.367, Z 7.650} C_DIS
   LIN {X -2.120, Y 8.356, Z 7.650} C_DIS
   LIN {X -2.065, Y 8.670, Z 7.650} C_DIS
   LIN {X -1.882, Y 9.844, Z 7.650} C_DIS
   LIN {X -1.717, Y 11.029, Z 7.650} C_DIS
   LIN {X -1.484, Y 13.152, Z 7.650} C_DIS
   LIN {X -1.391, Y 13.999, Z 7.650} C_DIS
   LIN {X -1.309, Y 15.009, Z 7.650} C_DIS
   LIN {X -1.247, Y 15.903, Z 7.650} C_DIS
   LIN {X -1.195, Y 16.817, Z 7.650} C_DIS
   LIN {X -1.152, Y 17.824, Z 7.650} C_DIS
   LIN {X -1.114, Y 19.292, Z 7.650} C_DIS
   LIN {X -1.113, Y 19.398, Z 7.650} C_DIS
   LIN {X -1.105, Y 20.788, Z 7.650} C_DIS
   LIN {X -1.116, Y 21.724, Z 7.650} C_DIS
   LIN {X -1.139, Y 22.658, Z 7.650} C_DIS
   LIN {X -1.145, Y 22.902, Z 7.650} C_DIS
   LIN {X -1.231, Y 24.775, Z 7.650} C_DIS
   LIN {X -1.297, Y 25.781, Z 7.650} C_DIS
   LIN {X -1.567, Y 28.669, Z 7.650} C_DIS
   LIN {X -1.583, Y 28.829, Z 7.650} C_DIS
   LIN {X -1.800, Y 30.538, Z 7.650} C_DIS
   LIN {X -1.818, Y 30.667, Z 7.650} C_DIS
   LIN {X -2.020, Y 32.017, Z 7.650} C_DIS
   LIN {X -2.288, Y 33.543, Z 7.650} C_DIS
   LIN {X -2.387, Y 34.112, Z 7.650} C_DIS
   LIN {X -2.455, Y 34.455, Z 7.650} C_DIS
   LIN {X -2.702, Y 35.682, Z 7.650} C_DIS
   LIN {X -2.943, Y 36.806, Z 7.650} C_DIS
   LIN {X -2.965, Y 36.906, Z 7.650} C_DIS
   LIN {X -2.976, Y 37.047, Z 7.650} C_DIS
   LIN {X -3.045, Y 38.279, Z 7.650} C_DIS
   LIN {X -2.707, Y 39.187, Z 7.650} C_DIS
   LIN {X -2.484, Y 39.896, Z 7.650} C_DIS
   LIN {X -2.042, Y 40.388, Z 7.650} C_DIS
   LIN {X -1.296, Y 41.122, Z 7.650} C_DIS
   LIN {X -0.573, Y 41.295, Z 7.650} C_DIS
   LIN {X 1.079, Y 41.779, Z 7.650} C_DIS
   LIN {X 2.683, Y 41.338, Z 7.650} C_DIS
   LIN {X 2.941, Y 41.167, Z 7.650} C_DIS
   LIN {X 4.095, Y 40.182, Z 7.650} C_DIS
   LIN {X 4.466, Y 39.437, Z 7.650} C_DIS
   LIN {X 4.751, Y 38.863, Z 7.650} C_DIS
   LIN {X 4.982, Y 38.041, Z 7.650} C_DIS
   LIN {X 5.154, Y 37.433, Z 7.650} C_DIS
   LIN {X 5.300, Y 36.886, Z 7.650} C_DIS
   LIN {X 5.646, Y 35.578, Z 7.650} C_DIS
   LIN {X 6.150, Y 33.516, Z 7.650} C_DIS
   LIN {X 6.214, Y 33.251, Z 7.650} C_DIS
   LIN {X 6.280, Y 32.955, Z 7.650} C_DIS
   LIN {X 6.579, Y 31.632, Z 7.650}
   LaserEnd_Ext()
   LIN {X 7.602, Y -2.377, Z 7.650}
   LaserStart_Ext()
   LIN {X 7.602, Y 18.604, Z 7.650}
   LaserEnd_Ext()
   LIN {X 6.602, Y 26.213, Z 7.650}
   LaserStart_Ext()
   LIN {X 6.602, Y -9.917, Z 7.650}
   LaserEnd_Ext()
   LIN {X 5.602, Y -15.097, Z 7.650}
   LaserStart_Ext()
   LIN {X 5.602, Y 31.419, Z 7.650}
   LaserEnd_Ext()
   LIN {X 4.602, Y 35.614, Z 7.650}
   LaserStart_Ext()
   LIN {X 4.602, Y -19.227, Z 7.650}
   LaserEnd_Ext()
   LIN {X 3.602, Y -22.858, Z 7.650}
   LaserStart_Ext()
   LIN {X 3.602, Y 38.929, Z 7.650}
   LaserEnd_Ext()
   LIN {X 2.602, Y 40.142, Z 7.650}
   LaserStart_Ext()
   LIN {X 2.602, Y -25.987, Z 7.650}
   LaserEnd_Ext()
   LIN {X 1.602, Y -27.922, Z 7.650}
   LaserStart_Ext()
   LIN {X 1.602, Y 40.599, Z 7.650}
   LaserEnd_Ext()
   LIN {X 0.602, Y 40.598, Z 7.650}
   LaserStart_Ext()
   LIN {X 0.602, Y -29.135, Z 7.650}
   LaserEnd_Ext()
   LIN {X -0.398, Y -29.982, Z 7.650}
   LaserStart_Ext()
   LIN {X -0.398, Y 13.883, Z 7.650}
   LaserEnd_Ext()
   LIN {X -0.398, Y 26.919, Z 7.650}
   LaserStart_Ext()
   LIN {X -0.398, Y 40.309, Z 7.650}
   LaserEnd_Ext()
   LIN {X -1.398, Y 39.608, Z 7.650}
   LaserStart_Ext()
   LIN {X -1.398, Y 34.264, Z 7.650}
   LaserEnd_Ext()
   LIN {X -1.398, Y 6.716, Z 7.650}
   LaserStart_Ext()
   LIN {X -1.398, Y -30.597, Z 7.650}
   LaserEnd_Ext()
   LIN {X -2.398, Y -30.943, Z 7.650}
   LaserStart_Ext()
   LIN {X -2.398, Y 2.239, Z 7.650}
   LaserEnd_Ext()
   LIN {X -3.398, Y -1.308, Z 7.650}
   LaserStart_Ext()
   LIN {X -3.398, Y -31.289, Z 7.650}
   LaserEnd_Ext()
   LIN {X -4.398, Y -31.404, Z 7.650}
   LaserStart_Ext()
   LIN {X -4.398, Y -4.312, Z 7.650}
   LaserEnd_Ext()
   LIN {X -5.398, Y -6.950, Z 7.650}
   LaserStart_Ext()
   LIN {X -5.398, Y -31.422, Z 7.650}
   LaserEnd_Ext()
   LIN {X -6.398, Y -31.344, Z 7.650}
   LaserStart_Ext()
   LIN {X -6.398, Y -9.263, Z 7.650}
   LaserEnd_Ext()
   LIN {X -7.398, Y -11.487, Z 7.650}
   LaserStart_Ext()
   LIN {X -7.398, Y -31.053, Z 7.650}
   LaserEnd_Ext()
   LIN {X -8.398, Y -30.717, Z 7.650}
   LaserStart_Ext()
   LIN {X -8.398, Y -13.448, Z 7.650}
   LaserEnd_Ext()
   LIN {X -9.398, Y -15.327, Z 7.650}
   LaserStart_Ext()
   LIN {X -9.398, Y -30.049, Z 7.650}
   LaserEnd_Ext()
   LIN {X -10.398, Y -29.298, Z 7.650}
   LaserStart_Ext()
   LIN {X -10.398, Y -17.069, Z 7.650}
   LaserEnd_Ext()
   LIN {X -11.398, Y -18.696, Z 7.650}
   LaserStart_Ext()
   LIN {X -11.398, Y -28.257, Z 7.650}
   LaserEnd_Ext()
   LIN {X -12.398, Y -26.487, Z 7.650}
   LaserStart_Ext()
   LIN {X -12.398, Y -20.792, Z 7.650}
   LaserEnd_Ext()
   LIN {X 9.056, Y 11.074, Z 8.500}
   LaserStart_Ext()
   LIN {X 9.101, Y 9.408, Z 8.500} C_DIS
   LIN {X 9.107, Y 8.363, Z 8.500} C_DIS
   LIN {X 9.111, Y 7.505, Z 8.500} C_DIS
   LIN {X 9.106, Y 6.878, Z 8.500} C_DIS
   LIN {X 9.095, Y 6.230, Z 8.500} C_DIS
   LIN {X 9.079, Y 5.624, Z 8.500} C_DIS
   LIN {X 9.048, Y 4.238, Z 8.500} C_DIS
   LIN {X 9.000, Y 3.024, Z 8.500} C_DIS
   LIN {X 8.963, Y 2.259, Z 8.500} C_DIS
   LIN {X 8.818, Y 0.021, Z 8.500} C_DIS
   LIN {X 8.668, Y -1.849, Z 8.500} C_DIS
   LIN {X 8.577, Y -2.872, Z 8.500} C_DIS
   LIN {X 8.528, Y -3.336, Z 8.500} C_DIS
   LIN {X 8.427, Y -4.230, Z 8.500} C_DIS
   LIN {X 8.335, Y -5.082, Z 8.500} C_DIS
   LIN {X 8.234, Y -5.882, Z 8.500} C_DIS
   LIN {X 8.127, Y -6.703, Z 8.500} C_DIS
   LIN {X 7.710, Y -9.507, Z 8.500} C_DIS
   LIN {X 6.913, Y -13.890, Z 8.500} C_DIS
   LIN {X 6.874, Y -14.110, Z 8.500} C_DIS
   LIN {X 6.838, Y -14.290, Z 8.500} C_DIS
   LIN {X 6.808, Y -14.434, Z 8.500} C_DIS
   LIN {X 6.763, Y -14.632, Z 8.500} C_DIS
   LIN {X 5.957, Y -18.193, Z 8.500} C_DIS
   LIN {X 5.744, Y -19.028, Z 8.500} C_DIS
   LIN {X 5.549, Y -19.760, Z 8.500} C_DIS
   LIN {X 4.958, Y -21.982, Z 8.500} C_DIS
   LIN {X 4.655, Y -23.030, Z 8.500} C_DIS
   LIN {X 4.259, Y -24.351, Z 8.500} C_DIS
   LIN {X 3.935, Y -25.372, Z 8.500} C_DIS
   LIN {X 3.673, Y -26.211, Z 8.500} C_DIS
   LIN {X 2.845, Y -27.657, Z 8.500} C_DIS
   LIN {X 2.198, Y -28.912, Z 8.500} C_DIS
   LIN {X 1.447, Y -29.786, Z 8.500} C_DIS
   LIN {X -0.451, Y -31.256, Z 8.500} C_DIS
   LIN {X -0.601, Y -31.357, Z 8.500} C_DIS
   LIN {X -1.156, Y -31.549, Z 8.500} C_DIS
   LIN {X -3.362, Y -32.330, Z 8.500} C_DIS
   LIN {X -4.567, Y -32.365, Z 8.500} C_DIS
   LIN {X -6.147, Y -32.394, Z 8.500} C_DIS
   LIN {X -7.441, Y -32.018, Z 8.500} C_DIS
   LIN {X -9.673, Y -31.076, Z 8.500} C_DIS
   LIN {X -11.003, Y -30.078, Z 8.500} C_DIS
   LIN {X -11.521, Y -29.614, Z 8.500} C_DIS
   LIN {X -11.974, Y -28.979, Z 8.500} C_DIS
   LIN {X -12.922, Y -27.614, Z 8.500} C_DIS
   LIN {X -13.166, Y -27.056, Z 8.500} C_DIS
   LIN {X -13.251, Y -26.516, Z 8.500} C_DIS
   LIN {X -13.876, Y -24.298, Z 8.500} C_DIS
   LIN {X -13.778, Y -22.451, Z 8.500} C_DIS
   LIN {X -13.621, Y -21.307, Z 8.500} C_DIS
   LIN {X -13.196, Y -20.376, Z 8.500} C_DIS
   LIN {X -12.500, Y -18.667, Z 8.500} C_DIS
   LIN {X -11.300, Y -16.687, Z 8.500} C_DIS
   LIN {X -10.930, Y -16.085, Z 8.500} C_DIS
   LIN {X -10.686, Y -15.664, Z 8.500} C_DIS
   LIN {X -9.354, Y -13.170, Z 8.500} C_DIS
   LIN {X -8.762, Y -12.052, Z 8.500} C_DIS
   LIN {X -8.583, Y -11.700, Z 8.500} C_DIS
   LIN {X -8.412, Y -11.349, Z 8.500} C_DIS
   LIN {X -8.243, Y -10.992, Z 8.500} C_DIS
   LIN {X -6.820, Y -7.788, Z 8.500} C_DIS
   LIN {X -6.422, Y -6.864, Z 8.500} C_DIS
   LIN {X -5.738, Y -5.060, Z 8.500} C_DIS
   LIN {X -5.581, Y -4.661, Z 8.500} C_DIS
   LIN {X -5.429, Y -4.258, Z 8.500} C_DIS
   LIN {X -5.285, Y -3.861, Z 8.500} C_DIS
   LIN {X -4.416, Y -1.213, Z 8.500} C_DIS
   LIN {X -4.369, Y -1.079, Z 8.500} C_DIS
   LIN {X -4.297, Y -0.858, Z 8.500} C_DIS
   LIN {X -4.205, Y -0.551, Z 8.500} C_DIS
   LIN {X -3.700, Y 1.215, Z 8.500} C_DIS
   LIN {X -3.371, Y 2.454, Z 8.500} C_DIS
   LIN {X -3.201, Y 3.136, Z 8.500} C_DIS
   LIN {X -3.057, Y 3.733, Z 8.500} C_DIS
   LIN {X -2.915, Y 4.355, Z 8.500} C_DIS
   LIN {X -2.813, Y 4.808, Z 8.500} C_DIS
   LIN {X -2.589, Y 5.875, Z 8.500} C_DIS
   LIN {X -2.559, Y 6.015, Z 8.500} C_DIS
   LIN {X -2.536, Y 6.133, Z 8.500} C_DIS
   LIN {X -2.320, Y 7.254, Z 8.500} C_DIS
   LIN {X -2.174, Y 8.100, Z 8.500} C_DIS
   LIN {X -2.063, Y 8.812, Z 8.500} C_DIS
   LIN {X -1.969, Y 9.502, Z 8.500} C_DIS
   LIN {X -1.793, Y 10.587, Z 8.500} C_DIS
   LIN {X -1.668, Y 11.581, Z 8.500} C_DIS
   LIN {X -1.456, Y 13.517, Z 8.500} C_DIS
   LIN {X -1.346, Y 14.947, Z 8.500} C_DIS
   LIN {X -1.298, Y 15.530, Z 8.500} C_DIS
   LIN {X -1.260, Y 16.078, Z 8.500} C_DIS
   LIN {X -1.228, Y 16.638, Z 8.500} C_DIS
   LIN {X -1.209, Y 17.069, Z 8.500} C_DIS
   LIN {X -1.184, Y 17.641, Z 8.500} C_DIS
   LIN {X -1.168, Y 18.177, Z 8.500} C_DIS
   LIN {X -1.146, Y 19.023, Z 8.500} C_DIS
   LIN {X -1.139, Y 19.664, Z 8.500} C_DIS
   LIN {X -1.135, Y 20.519, Z 8.500} C_DIS
   LIN {X -1.141, Y 21.095, Z 8.500} C_DIS
   LIN {X -1.156, Y 21.669, Z 8.500} C_DIS
   LIN {X -1.194, Y 23.254, Z 8.500} C_DIS
   LIN {X -1.247, Y 24.411, Z 8.500} C_DIS
   LIN {X -1.274, Y 24.882, Z 8.500} C_DIS
   LIN {X -1.313, Y 25.467, Z 8.500} C_DIS
   LIN {X -1.347, Y 25.928, Z 8.500} C_DIS
   LIN {X -1.514, Y 27.713, Z 8.500} C_DIS
   LIN {X -1.636, Y 28.909, Z 8.500} C_DIS
   LIN {X -1.773, Y 29.994, Z 8.500} C_DIS
   LIN {X -1.982, Y 31.441, Z 8.500} C_DIS
   LIN {X -2.052, Y 31.910, Z 8.500} C_DIS
   LIN {X -2.204, Y 32.779, Z 8.500} C_DIS
   LIN {X -2.449, Y 34.162, Z 8.500} C_DIS
   LIN {X -2.766, Y 35.719, Z 8.500} C_DIS
   LIN {X -3.033, Y 36.954, Z 8.500} C_DIS
   LIN {X -3.102, Y 37.830, Z 8.500} C_DIS
   LIN {X -3.129, Y 38.236, Z 8.500} C_DIS
   LIN {X -2.952, Y 38.827, Z 8.500} C_DIS
   LIN {X -2.648, Y 39.794, Z 8.500} C_DIS
   LIN {X -1.742, Y 40.803, Z 8.500} C_DIS
   LIN {X -1.526, Y 41.050, Z 8.500} C_DIS
   LIN {X -1.328, Y 41.155, Z 8.500} C_DIS
   LIN {X 1.003, Y 41.838, Z 8.500} C_DIS
   LIN {X 2.691, Y 41.377, Z 8.500} C_DIS
   LIN {X 3.674, Y 40.541, Z 8.500} C_DIS
   LIN {X 4.019, Y 40.247, Z 8.500} C_DIS
   LIN {X 4.269, Y 39.744, Z 8.500} C_DIS
   LIN {X 4.678, Y 38.930, Z 8.500} C_DIS
   LIN {X 4.862, Y 38.287, Z 8.500} C_DIS
   LIN {X 5.084, Y 37.501, Z 8.500} C_DIS
   LIN {X 5.488, Y 35.989, Z 8.500} C_DIS
   LIN {X 5.581, Y 35.641, Z 8.500} C_DIS
   LIN {X 5.643, Y 35.396, Z 8.500} C_DIS
   LIN {X 6.152, Y 33.331, Z 8.500} C_DIS
   LIN {X 6.378, Y 32.341, Z 8.500} C_DIS
   LIN {X 6.531, Y 31.666, Z 8.500} C_DIS
   LIN {X 6.592, Y 31.375, Z 8.500} C_DIS
   LIN {X 7.082, Y 28.939, Z 8.500} C_DIS
   LIN {X 7.198, Y 28.363, Z 8.500} C_DIS
   LIN {X 7.310, Y 27.784, Z 8.500} C_DIS
   LIN {X 7.411, Y 27.232, Z 8.500} C_DIS
   LIN {X 7.510, Y 26.661, Z 8.500} C_DIS
   LIN {X 7.652, Y 25.807, Z 8.500} C_DIS
   LIN {X 7.813, Y 24.790, Z 8.500} C_DIS
   LIN {X 8.138, Y 22.502, Z 8.500} C_DIS
   LIN {X 8.194, Y 22.105, Z 8.500} C_DIS
   LIN {X 8.246, Y 21.712, Z 8.500} C_DIS
   LIN {X 8.392, Y 20.452, Z 8.500} C_DIS
   LIN {X 8.497, Y 19.550, Z 8.500} C_DIS
   LIN {X 8.665, Y 17.800, Z 8.500} C_DIS
   LIN {X 8.691, Y 17.514, Z 8.500} C_DIS
   LIN {X 8.845, Y 15.591, Z 8.500} C_DIS
   LIN {X 8.886, Y 14.951, Z 8.500} C_DIS
   LIN {X 8.922, Y 14.311, Z 8.500} C_DIS
   LIN {X 8.952, Y 13.667, Z 8.500} C_DIS
   LIN {X 9.011, Y 12.622, Z 8.500} C_DIS
   LIN {X 9.031, Y 12.089, Z 8.500} C_DIS
   LIN {X 9.046, Y 11.575, Z 8.500} C_DIS
   LIN {X 9.056, Y 11.074, Z 8.500}
   LaserEnd_Ext()
   LIN {X 2.026, Y 40.522, Z 8.500}
   LaserStart_Ext()
   LIN {X 0.068, Y 40.522, Z 8.500}
   LaserEnd_Ext()
   LIN {X -1.548, Y 39.522, Z 8.500}
   LaserStart_Ext()
   LIN {X 3.263, Y 39.522, Z 8.500}
   LaserEnd_Ext()
   LIN {X 3.755, Y 38.522, Z 8.500}
   LaserStart_Ext()
   LIN {X -2.000, Y 38.522, Z 8.500}
   LaserEnd_Ext()
   LIN {X -2.075, Y 37.522, Z 8.500}
   LaserStart_Ext()
   LIN {X 4.039, Y 37.522, Z 8.500}
   LaserEnd_Ext()
   LIN {X 4.311, Y 36.522, Z 8.500}
   LaserStart_Ext()
   LIN {X -1.916, Y 36.522, Z 8.500}
   LaserEnd_Ext()
   LIN {X -1.705, Y 35.522, Z 8.500}
   LaserStart_Ext()
   LIN {X 4.578, Y 35.522, Z 8.500}
   LaserEnd_Ext()
   LIN {X 4.828, Y 34.522, Z 8.500}
   LaserStart_Ext()
   LIN {X -1.501, Y 34.522, Z 8.500}
   LaserEnd_Ext()
   LIN {X -1.320, Y 33.522, Z 8.500}
   LaserStart_Ext()
   LIN {X 5.075, Y 33.522, Z 8.500}
   LaserEnd_Ext()
   LIN {X 5.311, Y 32.522, Z 8.500}
   LaserStart_Ext()
   LIN {X -1.144, Y 32.522, Z 8.500}
   LaserEnd_Ext()
   LIN {X -0.983, Y 31.522, Z 8.500}
   LaserStart_Ext()
   LIN {X 5.538, Y 31.522, Z 8.500}
   LaserEnd_Ext()
   LIN {X 5.744, Y 30.522, Z 8.500}
   LaserStart_Ext()
   LIN {X -0.839, Y 30.522, Z 8.500}
   LaserEnd_Ext()
   LIN {X -0.705, Y 29.522, Z 8.500}
   LaserStart_Ext()
   LIN {X 5.945, Y 29.522, Z 8.500}
   LaserEnd_Ext()
   LIN {X 6.146, Y 28.522, Z 8.500}
   LaserStart_Ext()
   LIN {X -0.591, Y 28.522, Z 8.500}
   LaserEnd_Ext()
   LIN {X -0.492, Y 27.522, Z 8.500}
   LaserStart_Ext()
   LIN {X 6.341, Y 27.522, Z 8.500}
   LaserEnd_Ext()
   LIN {X 6.520, Y 26.522, Z 8.500}
   LaserStart_Ext()
   LIN {X -0.398, Y 26.522, Z 8.500}
   LaserEnd_Ext()
   LIN {X -0.315, Y 25.522, Z 8.500}
   LaserStart_Ext()
   LIN {X 6.684, Y 25.522, Z 8.500}
   LaserEnd_Ext()
   LIN {X 6.841, Y 24.522, Z 8.500}
   LaserStart_Ext()
   LIN {X -0.252, Y 24.522, Z 8.500}
   LaserEnd_Ext()
   LIN {X -0.206, Y 23.522, Z 8.500}
   LaserStart_Ext()
   LIN {X 6.983, Y 23.522, Z 8.500}
   LaserEnd_Ext()
   LIN {X 7.125, Y 22.522, Z 8.500}
   LaserStart_Ext()
   LIN {X -0.176, Y 22.522, Z 8.500}
   LaserEnd_Ext()
   LIN {X -0.152, Y 21.522, Z 8.500}
   LaserStart_Ext()
   LIN {X 7.261, Y 21.522, Z 8.500}
   LaserEnd_Ext()
   LIN {X 7.377, Y 20.522, Z 8.500}
   LaserStart_Ext()
   LIN {X -0.135, Y 20.522, Z 8.500}
   LaserEnd_Ext()
   LIN {X -0.141, Y 19.522, Z 8.500}
   LaserStart_Ext()
   LIN {X 7.493, Y 19.522, Z 8.500}
   LaserEnd_Ext()
   LIN {X 7.591, Y 18.522, Z 8.500}
   LaserStart_Ext()
   LIN {X -0.159, Y 18.522, Z 8.500}
   LaserEnd_Ext()
   LIN {X -0.189, Y 17.522, Z 8.500}
   LaserStart_Ext()
   LIN {X 7.686, Y 17.522, Z 8.500}
   LaserEnd_Ext()
   LIN {X 7.767, Y 16.522, Z 8.500}
   LaserStart_Ext()
   LIN {X -0.233, Y 16.522, Z 8.500}
   LaserEnd_Ext()
   LIN {X -0.296, Y 15.522, Z 8.500}
   LaserStart_Ext()
   LIN {X 7.847, Y 15.522, Z 8.500}
   LaserEnd_Ext()
   LIN {X 7.909, Y 14.522, Z 8.500}
   LaserStart_Ext()
   LIN {X -0.376, Y 14.522, Z 8.500}
   LaserEnd_Ext()
   LIN {X -0.453, Y 13.522, Z 8.500}
   LaserStart_Ext()
   LIN {X 7.959, Y 13.522, Z 8.500}
   LaserEnd_Ext()
   LIN {X 8.014, Y 12.522, Z 8.500}
   LaserStart_Ext()
   LIN {X -0.559, Y 12.522, Z 8.500}
   LaserEnd_Ext()
   LIN {X -0.669, Y 11.522, Z 8.500}
   LaserStart_Ext()
   LIN {X 8.047, Y 11.522, Z 8.500}
   LaserEnd_Ext()
   LIN {X 8.070, Y 10.522, Z 8.500}
   LaserStart_Ext()
   LIN {X -0.793, Y 10.522, Z 8.500}
   LaserEnd_Ext()
   LIN {X -0.952, Y 9.522, Z 8.500}
   LaserStart_Ext()
   LIN {X 8.097, Y 9.522, Z 8.500}
   LaserEnd_Ext()
   LIN {X 8.106, Y 8.522, Z 8.500}
   LaserStart_Ext()
   LIN {X -1.096, Y 8.522, Z 8.500}
   LaserEnd_Ext()
   LIN {X -1.259, Y 7.522, Z 8.500}
   LaserStart_Ext()
   LIN {X 8.110, Y 7.522, Z 8.500}
   LaserEnd_Ext()
   LIN {X 8.100, Y 6.522, Z 8.500}
   LaserStart_Ext()
   LIN {X -1.443, Y 6.522, Z 8.500}
   LaserEnd_Ext()
   LIN {X -1.641, Y 5.522, Z 8.500}
   LaserStart_Ext()
   LIN {X 8.077, Y 5.522, Z 8.500}
   LaserEnd_Ext()
   LIN {X 8.054, Y 4.522, Z 8.500}
   LaserStart_Ext()
   LIN {X -1.852, Y 4.522, Z 8.500}
   LaserEnd_Ext()
   LIN {X -2.079, Y 3.522, Z 8.500}
   LaserStart_Ext()
   LIN {X 8.019, Y 3.522, Z 8.500}
   LaserEnd_Ext()
   LIN {X 7.975, Y 2.522, Z 8.500}
   LaserStart_Ext()
   LIN {X -2.323, Y 2.522, Z 8.500}
   LaserEnd_Ext()
   LIN {X -2.584, Y 1.522, Z 8.500}
   LaserStart_Ext()
   LIN {X 7.914, Y 1.522, Z 8.500}
   LaserEnd_Ext()
   LIN {X 7.849, Y 0.522, Z 8.500}
   LaserStart_Ext()
   LIN {X -2.858, Y 0.522, Z 8.500}
   LaserEnd_Ext()
   LIN {X -3.144, Y -0.478, Z 8.500}
   LaserStart_Ext()
   LIN {X 7.775, Y -0.478, Z 8.500}
   LaserEnd_Ext()
   LIN {X 7.695, Y -1.478, Z 8.500}
   LaserStart_Ext()
   LIN {X -3.449, Y -1.478, Z 8.500}
   LaserEnd_Ext()
   LIN {X -3.779, Y -2.478, Z 8.500}
   LaserStart_Ext()
   LIN {X 7.608, Y -2.478, Z 8.500}
   LaserEnd_Ext()
   LIN {X 7.506, Y -3.478, Z 8.500}
   LaserStart_Ext()
   LIN {X -4.107, Y -3.478, Z 8.500}
   LaserEnd_Ext()
   LIN {X -4.445, Y -4.478, Z 8.500}
   LaserStart_Ext()
   LIN {X 7.394, Y -4.478, Z 8.500}
   LaserEnd_Ext()
   LIN {X 7.277, Y -5.478, Z 8.500}
   LaserStart_Ext()
   LIN {X -4.827, Y -5.478, Z 8.500}
   LaserEnd_Ext()
   LIN {X -5.206, Y -6.478, Z 8.500}
   LaserStart_Ext()
   LIN {X 7.148, Y -6.478, Z 8.500}
   LaserEnd_Ext()
   LIN {X 7.001, Y -7.478, Z 8.500}
   LaserStart_Ext()
   LIN {X -5.597, Y -7.478, Z 8.500}
   LaserEnd_Ext()
   LIN {X -6.032, Y -8.478, Z 8.500}
   LaserStart_Ext()
   LIN {X 6.852, Y -8.478, Z 8.500}
   LaserEnd_Ext()
   LIN {X 6.699, Y -9.478, Z 8.500}
   LaserStart_Ext()
   LIN {X -6.476, Y -9.478, Z 8.500}
   LaserEnd_Ext()
   LIN {X -6.921, Y -10.478, Z 8.500}
   LaserStart_Ext()
   LIN {X 6.517, Y -10.478, Z 8.500}
   LaserEnd_Ext()
   LIN {X 6.335, Y -11.478, Z 8.500}
   LaserStart_Ext()
   LIN {X -7.367, Y -11.478, Z 8.500}
   LaserEnd_Ext()
   LIN {X -7.857, Y -12.478, Z 8.500}
   LaserStart_Ext()
   LIN {X 6.153, Y -12.478, Z 8.500}
   LaserEnd_Ext()
   LIN {X 5.972, Y -13.478, Z 8.500}
   LaserStart_Ext()
   LIN {X -8.385, Y -13.478, Z 8.500}
   LaserEnd_Ext()
   LIN {X -8.919, Y -14.478, Z 8.500}
   LaserStart_Ext()
   LIN {X 5.773, Y -14.478, Z 8.500}
   LaserEnd_Ext()
   LIN {X 5.546, Y -15.478, Z 8.500}
   LaserStart_Ext()
   LIN {X -9.453, Y -15.478, Z 8.500}
   LaserEnd_Ext()
   LIN {X -10.002, Y -16.478, Z 8.500}
   LaserStart_Ext()
   LIN {X 5.320, Y -16.478, Z 8.500}
   LaserEnd_Ext()
   LIN {X 5.093, Y -17.478, Z 8.500}
   LaserStart_Ext()
   LIN {X -10.610, Y -17.478, Z 8.500}
   LaserEnd_Ext()
   LIN {X -11.216, Y -18.478, Z 8.500}
   LaserStart_Ext()
   LIN {X 4.852, Y -18.478, Z 8.500}
   LaserEnd_Ext()
   LIN {X 4.589, Y -19.478, Z 8.500}
   LaserStart_Ext()
   LIN {X -11.750, Y -19.478, Z 8.500}
   LaserEnd_Ext()
   LIN {X -12.158, Y -20.478, Z 8.500}
   LaserStart_Ext()
   LIN {X 4.323, Y -20.478, Z 8.500}
   LaserEnd_Ext()
   LIN {X 4.057, Y -21.478, Z 8.500}
   LaserStart_Ext()
   LIN {X -12.600, Y -21.478, Z 8.500}
   LaserEnd_Ext()
   LIN {X -12.772, Y -22.478, Z 8.500}
   LaserStart_Ext()
   LIN {X 3.774, Y -22.478, Z 8.500}
   LaserEnd_Ext()
   LIN {X 3.477, Y -23.478, Z 8.500}
   LaserStart_Ext()
   LIN {X -12.831, Y -23.478, Z 8.500}
   LaserEnd_Ext()
   LIN {X -12.786, Y -24.478, Z 8.500}
   LaserStart_Ext()
   LIN {X 3.170, Y -24.478, Z 8.500}
   LaserEnd_Ext()
   LIN {X 2.855, Y -25.478, Z 8.500}
   LaserStart_Ext()
   LIN {X -12.504, Y -25.478, Z 8.500}
   LaserEnd_Ext()
   LIN {X -12.245, Y -26.478, Z 8.500}
   LaserStart_Ext()
   LIN {X 2.368, Y -26.478, Z 8.500}
   LaserEnd_Ext()
   LIN {X 1.812, Y -27.478, Z 8.500}
   LaserStart_Ext()
   LIN {X -11.799, Y -27.478, Z 8.500}
   LaserEnd_Ext()
   LIN {X -11.103, Y -28.478, Z 8.500}
   LaserStart_Ext()
   LIN {X 1.252, Y -28.478, Z 8.500}
   LaserEnd_Ext()
   LIN {X 0.211, Y -29.478, Z 8.500}
   LaserStart_Ext()
   LIN {X -10.136, Y -29.478, Z 8.500}
   LaserEnd_Ext()
   LIN {X -8.517, Y -30.478, Z 8.500}
   LaserStart_Ext()
   LIN {X -1.120, Y -30.478, Z 8.500}
   LaserEnd_Ext()
   LIN {X -5.059, Y -23.621, Z 9.350}
   LaserStart_Ext()
   LIN {X -5.136, Y -23.483, Z 9.350} C_DIS
   LIN {X -5.135, Y -23.313, Z 9.350} C_DIS
   LIN {X -5.065, Y -23.221, Z 9.350} C_DIS
   LIN {X -4.989, Y -23.123, Z 9.350} C_DIS
   LIN {X -4.887, Y -23.092, Z 9.350} C_DIS
   LIN {X -4.702, Y -23.108, Z 9.350} C_DIS
   LIN {X -4.590, Y -23.181, Z 9.350} C_DIS
   LIN {X -4.518, Y -23.309, Z 9.350} C_DIS
   LIN {X -4.515, Y -23.431, Z 9.350} C_DIS
   LIN {X -4.580, Y -23.600, Z 9.350} C_DIS
   LIN {X -4.696, Y -23.689, Z 9.350} C_DIS
   LIN {X -4.823, Y -23.718, Z 9.350} C_DIS
   LIN {X -4.969, Y -23.687, Z 9.350} C_DIS
   LIN {X -5.050, Y -23.628, Z 9.350} C_DIS
   LIN {X -5.059, Y -23.621, Z 9.350}
   LaserEnd_Ext()
   LIN {X -1.329, Y 25.154, Z 9.350}
   LaserStart_Ext()
   LIN {X -1.392, Y 26.008, Z 9.350} C_DIS
   LIN {X -1.462, Y 26.758, Z 9.350} C_DIS
   LIN {X -1.688, Y 28.988, Z 9.350} C_DIS
   LIN {X -1.747, Y 29.449, Z 9.350} C_DIS
   LIN {X -1.936, Y 30.765, Z 9.350} C_DIS
   LIN {X -2.095, Y 31.877, Z 9.350} C_DIS
   LIN {X -2.401, Y 33.597, Z 9.350} C_DIS
   LIN {X -2.510, Y 34.212, Z 9.350} C_DIS
   LIN {X -2.555, Y 34.435, Z 9.350} C_DIS
   LIN {X -2.833, Y 35.780, Z 9.350} C_DIS
   LIN {X -3.037, Y 36.716, Z 9.350} C_DIS
   LIN {X -3.101, Y 37.003, Z 9.350} C_DIS
   LIN {X -3.123, Y 37.395, Z 9.350} C_DIS
   LIN {X -3.189, Y 38.383, Z 9.350} C_DIS
   LIN {X -2.936, Y 39.226, Z 9.350} C_DIS
   LIN {X -2.735, Y 39.824, Z 9.350} C_DIS
   LIN {X -2.045, Y 40.618, Z 9.350} C_DIS
   LIN {X -1.485, Y 41.205, Z 9.350} C_DIS
   LIN {X -0.296, Y 41.538, Z 9.350} C_DIS
   LIN {X 0.924, Y 41.895, Z 9.350} C_DIS
   LIN {X 2.242, Y 41.540, Z 9.350} C_DIS
   LIN {X 2.612, Y 41.439, Z 9.350} C_DIS
   LIN {X 3.004, Y 41.106, Z 9.350} C_DIS
   LIN {X 3.944, Y 40.312, Z 9.350} C_DIS
   LIN {X 4.351, Y 39.505, Z 9.350} C_DIS
   LIN {X 4.606, Y 38.996, Z 9.350} C_DIS
   LIN {X 4.825, Y 38.229, Z 9.350} C_DIS
   LIN {X 5.019, Y 37.555, Z 9.350} C_DIS
   LIN {X 5.164, Y 37.022, Z 9.350} C_DIS
   LIN {X 5.527, Y 35.674, Z 9.350} C_DIS
   LIN {X 6.016, Y 33.710, Z 9.350} C_DIS
   LIN {X 6.101, Y 33.365, Z 9.350} C_DIS
   LIN {X 6.228, Y 32.812, Z 9.350} C_DIS
   LIN {X 6.437, Y 31.901, Z 9.350} C_DIS
   LIN {X 6.510, Y 31.583, Z 9.350} C_DIS
   LIN {X 6.761, Y 30.305, Z 9.350} C_DIS
   LIN {X 7.262, Y 27.809, Z 9.350} C_DIS
   LIN {X 7.323, Y 27.509, Z 9.350} C_DIS
   LIN {X 7.381, Y 27.207, Z 9.350} C_DIS
   LIN {X 7.434, Y 26.919, Z 9.350} C_DIS
   LIN {X 7.486, Y 26.622, Z 9.350} C_DIS
   LIN {X 7.724, Y 25.180, Z 9.350} C_DIS
   LIN {X 8.235, Y 21.592, Z 9.350} C_DIS
   LIN {X 8.261, Y 21.405, Z 9.350} C_DIS
   LIN {X 8.296, Y 21.105, Z 9.350} C_DIS
   LIN {X 8.488, Y 19.454, Z 9.350} C_DIS
   LIN {X 8.584, Y 18.455, Z 9.350} C_DIS
   LIN {X 8.750, Y 16.598, Z 9.350} C_DIS
   LIN {X 8.843, Y 15.433, Z 9.350} C_DIS
   LIN {X 8.868, Y 15.045, Z 9.350} C_DIS
   LIN {X 8.890, Y 14.657, Z 9.350} C_DIS
   LIN {X 8.908, Y 14.267, Z 9.350} C_DIS
   LIN {X 9.009, Y 12.460, Z 9.350} C_DIS
   LIN {X 9.016, Y 12.283, Z 9.350} C_DIS
   LIN {X 9.021, Y 12.112, Z 9.350} C_DIS
   LIN {X 9.024, Y 11.945, Z 9.350} C_DIS
   LIN {X 9.102, Y 9.054, Z 9.350} C_DIS
   LIN {X 9.104, Y 8.738, Z 9.350} C_DIS
   LIN {X 9.110, Y 7.237, Z 9.350} C_DIS
   LIN {X 9.107, Y 6.899, Z 9.350} C_DIS
   LIN {X 9.101, Y 6.550, Z 9.350} C_DIS
   LIN {X 9.093, Y 6.224, Z 9.350} C_DIS
   LIN {X 9.038, Y 3.791, Z 9.350} C_DIS
   LIN {X 9.013, Y 3.153, Z 9.350} C_DIS
   LIN {X 8.949, Y 1.811, Z 9.350} C_DIS
   LIN {X 8.873, Y 0.639, Z 9.350} C_DIS
   LIN {X 8.577, Y -3.048, Z 9.350} C_DIS
   LIN {X 8.365, Y -5.012, Z 9.350} C_DIS
   LIN {X 8.295, Y -5.566, Z 9.350} C_DIS
   LIN {X 8.051, Y -7.443, Z 9.350} C_DIS
   LIN {X 7.817, Y -9.015, Z 9.350} C_DIS
   LIN {X 7.282, Y -11.956, Z 9.350} C_DIS
   LIN {X 6.942, Y -13.932, Z 9.350} C_DIS
   LIN {X 6.739, Y -14.939, Z 9.350} C_DIS
   LIN {X 5.930, Y -18.487, Z 9.350} C_DIS
   LIN {X 5.753, Y -19.197, Z 9.350} C_DIS
   LIN {X 5.054, Y -21.829, Z 9.350} C_DIS
   LIN {X 4.461, Y -23.882, Z 9.350} C_DIS
   LIN {X 4.339, Y -24.288, Z 9.350} C_DIS
   LIN {X 4.240, Y -24.601, Z 9.350} C_DIS
   LIN {X 3.756, Y -26.149, Z 9.350} C_DIS
   LIN {X 2.228, Y -28.817, Z 9.350} C_DIS
   LIN {X 2.022, Y -29.216, Z 9.350} C_DIS
   LIN {X 1.784, Y -29.494, Z 9.350} C_DIS
   LIN {X 0.971, Y -30.123, Z 9.350} C_DIS
   LIN {X -0.469, Y -31.283, Z 9.350} C_DIS
   LIN {X -1.261, Y -31.583, Z 9.350} C_DIS
   LIN {X -3.212, Y -32.274, Z 9.350} C_DIS
   LIN {X -5.571, Y -32.341, Z 9.350} C_DIS
   LIN {X -6.078, Y -32.350, Z 9.350} C_DIS
   LIN {X -6.493, Y -32.230, Z 9.350} C_DIS
   LIN {X -10.194, Y -30.668, Z 9.350} C_DIS
   LIN {X -10.472, Y -30.459, Z 9.350} C_DIS
   LIN {X -11.326, Y -29.695, Z 9.350} C_DIS
   LIN {X -11.584, Y -29.333, Z 9.350} C_DIS
   LIN {X -12.620, Y -27.842, Z 9.350} C_DIS
   LIN {X -12.920, Y -27.431, Z 9.350} C_DIS
   LIN {X -13.044, Y -27.038, Z 9.350} C_DIS
   LIN {X -13.783, Y -24.412, Z 9.350} C_DIS
   LIN {X -13.635, Y -21.607, Z 9.350} C_DIS
   LIN {X -12.435, Y -18.643, Z 9.350} C_DIS
   LIN {X -11.089, Y -16.421, Z 9.350} C_DIS
   LIN {X -10.786, Y -15.912, Z 9.350} C_DIS
   LIN {X -10.242, Y -14.881, Z 9.350} C_DIS
   LIN {X -9.016, Y -12.586, Z 9.350} C_DIS
   LIN {X -8.676, Y -11.944, Z 9.350} C_DIS
   LIN {X -8.573, Y -11.741, Z 9.350} C_DIS
   LIN {X -8.475, Y -11.540, Z 9.350} C_DIS
   LIN {X -8.378, Y -11.335, Z 9.350} C_DIS
   LIN {X -6.562, Y -7.248, Z 9.350} C_DIS
   LIN {X -6.497, Y -7.098, Z 9.350} C_DIS
   LIN {X -5.369, Y -4.120, Z 9.350} C_DIS
   LIN {X -5.302, Y -3.943, Z 9.350} C_DIS
   LIN {X -4.160, Y -0.394, Z 9.350} C_DIS
   LIN {X -3.870, Y 0.627, Z 9.350} C_DIS
   LIN {X -3.610, Y 1.537, Z 9.350} C_DIS
   LIN {X -3.485, Y 2.007, Z 9.350} C_DIS
   LIN {X -3.160, Y 3.308, Z 9.350} C_DIS
   LIN {X -3.101, Y 3.554, Z 9.350} C_DIS
   LIN {X -2.866, Y 4.587, Z 9.350} C_DIS
   LIN {X -2.758, Y 5.111, Z 9.350} C_DIS
   LIN {X -2.423, Y 6.757, Z 9.350} C_DIS
   LIN {X -2.349, Y 7.141, Z 9.350} C_DIS
   LIN {X -2.309, Y 7.376, Z 9.350} C_DIS
   LIN {X -2.278, Y 7.574, Z 9.350} C_DIS
   LIN {X -2.252, Y 7.765, Z 9.350} C_DIS
   LIN {X -1.879, Y 10.060, Z 9.350} C_DIS
   LIN {X -1.616, Y 12.162, Z 9.350} C_DIS
   LIN {X -1.521, Y 13.035, Z 9.350} C_DIS
   LIN {X -1.305, Y 15.836, Z 9.350} C_DIS
   LIN {X -1.287, Y 16.051, Z 9.350} C_DIS
   LIN {X -1.273, Y 16.252, Z 9.350} C_DIS
   LIN {X -1.261, Y 16.458, Z 9.350} C_DIS
   LIN {X -1.226, Y 17.247, Z 9.350} C_DIS
   LIN {X -1.217, Y 17.458, Z 9.350} C_DIS
   LIN {X -1.187, Y 18.439, Z 9.350} C_DIS
   LIN {X -1.179, Y 18.754, Z 9.350} C_DIS
   LIN {X -1.166, Y 19.929, Z 9.350} C_DIS
   LIN {X -1.164, Y 20.249, Z 9.350} C_DIS
   LIN {X -1.167, Y 20.465, Z 9.350} C_DIS
   LIN {X -1.172, Y 20.680, Z 9.350} C_DIS
   LIN {X -1.243, Y 23.606, Z 9.350} C_DIS
   LIN {X -1.263, Y 24.046, Z 9.350} C_DIS
   LIN {X -1.314, Y 24.920, Z 9.350} C_DIS
   LIN {X -1.329, Y 25.154, Z 9.350}
   LaserEnd_Ext()
   LIN {X -12.280, Y -20.911, Z 9.350}
   LaserStart_Ext()
   LIN {X -12.280, Y -26.062, Z 9.350}
   LaserEnd_Ext()
   LIN {X -11.280, Y -28.018, Z 9.350}
   LaserStart_Ext()
   LIN {X -11.280, Y -18.667, Z 9.350}
   LaserEnd_Ext()
   LIN {X -10.280, Y -17.016, Z 9.350}
   LaserStart_Ext()
   LIN {X -10.280, Y -29.289, Z 9.350}
   LaserEnd_Ext()
   LIN {X -9.280, Y -29.968, Z 9.350}
   LaserStart_Ext()
   LIN {X -9.280, Y -15.203, Z 9.350}
   LaserEnd_Ext()
   LIN {X -8.280, Y -13.331, Z 9.350}
   LaserStart_Ext()
   LIN {X -8.280, Y -30.390, Z 9.350}
   LaserEnd_Ext()
   LIN {X -7.280, Y -30.812, Z 9.350}
   LaserStart_Ext()
   LIN {X -7.280, Y -11.327, Z 9.350}
   LaserEnd_Ext()
   LIN {X -6.280, Y -9.076, Z 9.350}
   LaserStart_Ext()
   LIN {X -6.280, Y -31.234, Z 9.350}
   LaserEnd_Ext()
   LIN {X -5.280, Y -31.332, Z 9.350}
   LaserStart_Ext()
   LIN {X -5.280, Y -24.637, Z 9.350}
   LaserEnd_Ext()
   LIN {X -5.280, Y -22.166, Z 9.350}
   LaserStart_Ext()
   LIN {X -5.280, Y -6.708, Z 9.350}
   LaserEnd_Ext()
   LIN {X -4.280, Y -4.031, Z 9.350}
   LaserStart_Ext()
   LIN {X -4.280, Y -22.196, Z 9.350}
   LaserEnd_Ext()
   LIN {X -4.280, Y -24.598, Z 9.350}
   LaserStart_Ext()
   LIN {X -4.280, Y -31.304, Z 9.350}
   LaserEnd_Ext()
   LIN {X -3.280, Y -31.237, Z 9.350}
   LaserStart_Ext()
   LIN {X -3.280, Y -0.924, Z 9.350}
   LaserEnd_Ext()
   LIN {X -2.280, Y 2.705, Z 9.350}
   LaserStart_Ext()
   LIN {X -2.280, Y -30.882, Z 9.350}
   LaserEnd_Ext()
   LIN {X -1.280, Y -30.520, Z 9.350}
   LaserStart_Ext()
   LIN {X -1.280, Y 7.492, Z 9.350}
   LaserEnd_Ext()
   LIN {X -1.280, Y 33.004, Z 9.350}
   LaserStart_Ext()
   LIN {X -1.280, Y 39.971, Z 9.350}
   LaserEnd_Ext()
   LIN {X -0.280, Y 40.504, Z 9.350}
   LaserStart_Ext()
   LIN {X -0.280, Y 24.360, Z 9.350}
   LaserEnd_Ext()
   LIN {X -0.280, Y 16.121, Z 9.350}
   LaserStart_Ext()
   LIN {X -0.280, Y -29.847, Z 9.350}
   LaserEnd_Ext()
   LIN {X 0.720, Y -29.053, Z 9.350}
   LaserStart_Ext()
   LIN {X 0.720, Y 40.793, Z 9.350}
   LaserEnd_Ext()
   LIN {X 1.720, Y 40.645, Z 9.350}
   LaserStart_Ext()
   LIN {X 1.720, Y -27.692, Z 9.350}
   LaserEnd_Ext()
   LIN {X 2.720, Y -25.945, Z 9.350}
   LaserStart_Ext()
   LIN {X 2.720, Y 40.037, Z 9.350}
   LaserEnd_Ext()
   LIN {X 3.720, Y 38.458, Z 9.350}
   LaserStart_Ext()
   LIN {X 3.720, Y -22.842, Z 9.350}
   LaserEnd_Ext()
   LIN {X 4.720, Y -19.191, Z 9.350}
   LaserStart_Ext()
   LIN {X 4.720, Y 34.775, Z 9.350}
   LaserEnd_Ext()
   LIN {X 5.720, Y 30.415, Z 9.350}
   LaserStart_Ext()
   LIN {X 5.720, Y -14.910, Z 9.350}
   LaserEnd_Ext()
   LIN {X 6.720, Y -9.456, Z 9.350}
   LaserStart_Ext()
   LIN {X 6.720, Y 25.122, Z 9.350}
   LaserEnd_Ext()
   LIN {X 7.720, Y 16.885, Z 9.350}
   LaserStart_Ext()
   LIN {X 7.720, Y -1.225, Z 9.350}
   LaserEnd_Ext()
   LIN {X -4.185, Y -22.252, Z 10.200}
   LaserStart_Ext()
   LIN {X -3.899, Y -22.463, Z 10.200} C_DIS
   LIN {X -3.803, Y -22.584, Z 10.200} C_DIS
   LIN {X -3.686, Y -22.758, Z 10.200} C_DIS
   LIN {X -3.637, Y -22.919, Z 10.200} C_DIS
   LIN {X -3.671, Y -23.171, Z 10.200} C_DIS
   LIN {X -3.671, Y -23.779, Z 10.200} C_DIS
   LIN {X -3.822, Y -24.015, Z 10.200} C_DIS
   LIN {X -3.953, Y -24.167, Z 10.200} C_DIS
   LIN {X -4.275, Y -24.362, Z 10.200} C_DIS
   LIN {X -4.404, Y -24.423, Z 10.200} C_DIS
   LIN {X -4.819, Y -24.456, Z 10.200} C_DIS
   LIN {X -4.926, Y -24.457, Z 10.200} C_DIS
   LIN {X -5.257, Y -24.357, Z 10.200} C_DIS
   LIN {X -5.491, Y -24.169, Z 10.200} C_DIS
   LIN {X -5.677, Y -24.009, Z 10.200} C_DIS
   LIN {X -5.819, Y -23.723, Z 10.200} C_DIS
   LIN {X -5.887, Y -23.505, Z 10.200} C_DIS
   LIN {X -5.901, Y -23.173, Z 10.200} C_DIS
   LIN {X -5.857, Y -22.980, Z 10.200} C_DIS
   LIN {X -5.601, Y -22.551, Z 10.200} C_DIS
   LIN {X -5.497, Y -22.406, Z 10.200} C_DIS
   LIN {X -5.300, Y -22.292, Z 10.200} C_DIS
   LIN {X -5.086, Y -22.175, Z 10.200} C_DIS
   LIN {X -4.788, Y -22.147, Z 10.200} C_DIS
   LIN {X -4.616, Y -22.124, Z 10.200} C_DIS
   LIN {X -4.196, Y -22.246, Z 10.200} C_DIS
   LIN {X -4.185, Y -22.252, Z 10.200}
   LaserEnd_Ext()
   LIN {X -4.877, Y -2.572, Z 10.200}
   LaserStart_Ext()
   LIN {X -4.013, Y 0.112, Z 10.200} C_DIS
   LIN {X -3.554, Y 1.731, Z 10.200} C_DIS
   LIN {X -3.168, Y 3.278, Z 10.200} C_DIS
   LIN {X -3.019, Y 3.950, Z 10.200} C_DIS
   LIN {X -2.555, Y 6.217, Z 10.200} C_DIS
   LIN {X -2.381, Y 7.007, Z 10.200} C_DIS
   LIN {X -2.191, Y 8.149, Z 10.200} C_DIS
   LIN {X -1.966, Y 9.533, Z 10.200} C_DIS
   LIN {X -1.674, Y 11.869, Z 10.200} C_DIS
   LIN {X -1.580, Y 12.607, Z 10.200} C_DIS
   LIN {X -1.569, Y 12.742, Z 10.200} C_DIS
   LIN {X -1.293, Y 16.277, Z 10.200} C_DIS
   LIN {X -1.286, Y 16.440, Z 10.200} C_DIS
   LIN {X -1.245, Y 17.343, Z 10.200} C_DIS
   LIN {X -1.211, Y 18.471, Z 10.200} C_DIS
   LIN {X -1.196, Y 19.830, Z 10.200} C_DIS
   LIN {X -1.195, Y 20.242, Z 10.200} C_DIS
   LIN {X -1.279, Y 23.670, Z 10.200} C_DIS
   LIN {X -1.340, Y 24.735, Z 10.200} C_DIS
   LIN {X -1.419, Y 25.823, Z 10.200} C_DIS
   LIN {X -1.432, Y 26.051, Z 10.200} C_DIS
   LIN {X -1.452, Y 26.225, Z 10.200} C_DIS
   LIN {X -1.483, Y 26.534, Z 10.200} C_DIS
   LIN {X -1.740, Y 29.061, Z 10.200} C_DIS
   LIN {X -1.887, Y 30.083, Z 10.200} C_DIS
   LIN {X -2.150, Y 31.927, Z 10.200} C_DIS
   LIN {X -2.300, Y 32.773, Z 10.200} C_DIS
   LIN {X -2.570, Y 34.262, Z 10.200} C_DIS
   LIN {X -2.881, Y 35.756, Z 10.200} C_DIS
   LIN {X -2.922, Y 35.943, Z 10.200} C_DIS
   LIN {X -3.167, Y 37.051, Z 10.200} C_DIS
   LIN {X -3.228, Y 38.135, Z 10.200} C_DIS
   LIN {X -3.247, Y 38.525, Z 10.200} C_DIS
   LIN {X -3.065, Y 39.048, Z 10.200} C_DIS
   LIN {X -2.759, Y 39.961, Z 10.200} C_DIS
   LIN {X -2.564, Y 40.185, Z 10.200} C_DIS
   LIN {X -1.507, Y 41.294, Z 10.200} C_DIS
   LIN {X 0.735, Y 41.921, Z 10.200} C_DIS
   LIN {X 0.845, Y 41.953, Z 10.200} C_DIS
   LIN {X 1.051, Y 41.897, Z 10.200} C_DIS
   LIN {X 2.535, Y 41.501, Z 10.200} C_DIS
   LIN {X 3.315, Y 40.846, Z 10.200} C_DIS
   LIN {X 3.869, Y 40.378, Z 10.200} C_DIS
   LIN {X 4.182, Y 39.758, Z 10.200} C_DIS
   LIN {X 4.535, Y 39.063, Z 10.200} C_DIS
